LIN {X 0,Y 529.765,Z 572.438,A -85,B 0,C 180,E1 25488.601,E2 25488.601} C_VEL
LIN {X 0,Y 529.183,Z 585.576,A -85,B 0,C 180,E1 25486.804,E2 25486.804} C_VEL
LIN {X 0,Y 528.717,Z 597.375,A -85,B 0,C 180,E1 25484.904,E2 25484.904} C_VEL
LIN {X 0,Y 528.358,Z 608.331,A -85,B 0,C 180,E1 25482.792,E2 25482.792} C_VEL
LIN {X 0,Y 528.139,Z 617.247,A -85,B 0,C 180,E1 25480.693,E2 25480.693} C_VEL
LIN {X 0,Y 528.011,Z 624.374,A -85,B 0,C 180,E1 25478.604,E2 25478.604} C_VEL
LIN {X 0,Y 527.933,Z 630.003,A -85,B 0,C 180,E1 25476.416,E2 25476.416} C_VEL
LIN {X 0,Y 527.91,Z 633.928,A -85,B 0,C 180,E1 25474.237,E2 25474.237} C_VEL
LIN {X 0,Y 527.911,Z 636.306,A -85,B 0,C 180,E1 25471.954,E2 25471.954} C_VEL
LIN {X 0,Y 527.906,Z 636.962,A -85,B 0,C 180,E1 25469.784,E2 25469.784} C_VEL
LIN {X 0,Y 527.901,Z 636.034,A -85,B 0,C 180,E1 25467.613,E2 25467.613} C_VEL
LIN {X 0,Y 527.913,Z 633.45,A -85,B 0,C 180,E1 25465.438,E2 25465.438} C_VEL
LIN {X 0,Y 527.952,Z 629.246,A -85,B 0,C 180,E1 25463.258,E2 25463.258} C_VEL
LIN {X 0,Y 528.029,Z 623.329,A -85,B 0,C 180,E1 25461.068,E2 25461.068} C_VEL
LIN {X 0,Y 528.171,Z 616.015,A -85,B 0,C 180,E1 25458.978,E2 25458.978} C_VEL
LIN {X 0,Y 528.406,Z 606.785,A -85,B 0,C 180,E1 25456.876,E2 25456.876} C_VEL
LIN {X 0,Y 528.766,Z 596.111,A -85,B 0,C 180,E1 25454.874,E2 25454.874} C_VEL
LIN {X 0,Y 529.254,Z 583.72,A -85,B 0,C 180,E1 25452.926,E2 25452.926} C_VEL
LIN {X 0,Y 529.883,Z 569.672,A -85,B 0,C 180,E1 25451.062,E2 25451.062} C_VEL
LIN {X 0,Y 530.615,Z 554.618,A -85,B 0,C 180,E1 25449.368,E2 25449.368} C_VEL
LIN {X 0,Y 531.432,Z 538.622,A -85,B 0,C 180,E1 25447.839,E2 25447.839} C_VEL
LIN {X 0,Y 532.324,Z 520.994,A -85,B 0,C 180,E1 25446.418,E2 25446.418} C_VEL
LIN {X 0,Y 533.203,Z 502.232,A -85,B 0,C 180,E1 25445.164,E2 25445.164} C_VEL
LIN {X 0,Y 534.026,Z 483.351,A -85,B 0,C 180,E1 25444.136,E2 25444.136} C_VEL
LIN {X 0,Y 534.767,Z 464.127,A -85,B 0,C 180,E1 25443.301,E2 25443.301} C_VEL
LIN {X 0,Y 535.396,Z 443.369,A -85,B 0,C 180,E1 25442.614,E2 25442.614} C_VEL
LIN {X 0,Y 535.876,Z 422.691,A -85,B 0,C 180,E1 25442.142,E2 25442.142} C_VEL
LIN {X 0,Y 537.477,Z 229.841,A -85,B 0,C 180,E1 25439.341,E2 25439.341} C_VEL
LIN {X 0,Y 537.719,Z 174.211,A -85,B 0,C 180,E1 25438.529,E2 25438.529} C_VEL
LIN {X 0,Y 535.937,Z 162.685,A -85,B 0,C 180,E1 25438.227,E2 25438.227} C_VEL
LIN {X 0,Y 536.978,Z 125.392,A -85,B 0,C 180,E1 25435.72,E2 25435.72} C_VEL
LIN {X 0,Y 528.489,Z 103.658,A -85,B 0,C 180,E1 25433.555,E2 25433.555} C_VEL
LIN {X 0,Y 528.528,Z 103.65,A -85,B 0,C 180,E1 25430.18,E2 25430.18} C_VEL
LIN {X 0,Y 528.47,Z 103.654,A -85,B 0,C 180,E1 25426.912,E2 25426.912} C_VEL
LIN {X 0,Y 528.472,Z 103.65,A -85,B 0,C 180,E1 25423.406,E2 25423.406} C_VEL
LIN {X 0,Y 528.528,Z 103.639,A -85,B 0,C 180,E1 25420.159,E2 25420.159} C_VEL
LIN {X 0,Y 528.473,Z 103.643,A -85,B 0,C 180,E1 25416.842,E2 25416.842} C_VEL
LIN {X 0,Y 528.467,Z 103.648,A -85,B 0,C 180,E1 25413.406,E2 25413.406} C_VEL
LIN {X 0,Y 528.522,Z 103.651,A -85,B 0,C 180,E1 25410.088,E2 25410.088} C_VEL
LIN {X 0,Y 528.482,Z 103.651,A -85,B 0,C 180,E1 25406.75,E2 25406.75} C_VEL
LIN {X 0,Y 528.463,Z 103.649,A -85,B 0,C 180,E1 25403.411,E2 25403.411} C_VEL
LIN {X 0,Y 528.514,Z 103.648,A -85,B 0,C 180,E1 25400.14,E2 25400.14} C_VEL
LIN {X 0,Y 528.482,Z 103.65,A -85,B 0,C 180,E1 25396.803,E2 25396.803} C_VEL
LIN {X 0,Y 528.459,Z 103.644,A -85,B 0,C 180,E1 25393.457,E2 25393.457} C_VEL
LIN {X 0,Y 528.504,Z 103.654,A -85,B 0,C 180,E1 25390.133,E2 25390.133} C_VEL
LIN {X 0,Y 528.479,Z 103.643,A -85,B 0,C 180,E1 25386.845,E2 25386.845} C_VEL
LIN {X 0,Y 528.457,Z 103.653,A -85,B 0,C 180,E1 25383.471,E2 25383.471} C_VEL
LIN {X 0,Y 528.491,Z 103.65,A -85,B 0,C 180,E1 25380.108,E2 25380.108} C_VEL
LIN {X 0,Y 528.483,Z 103.653,A -85,B 0,C 180,E1 25376.855,E2 25376.855} C_VEL
LIN {X 0,Y 528.453,Z 103.65,A -85,B 0,C 180,E1 25373.59,E2 25373.59} C_VEL
LIN {X 0,Y 528.503,Z 103.65,A -85,B 0,C 180,E1 25370.306,E2 25370.306} C_VEL
LIN {X 0,Y 528.474,Z 103.648,A -85,B 0,C 180,E1 25366.988,E2 25366.988} C_VEL
LIN {X 0,Y 528.451,Z 103.65,A -85,B 0,C 180,E1 25363.625,E2 25363.625} C_VEL
LIN {X 0,Y 528.496,Z 103.655,A -85,B 0,C 180,E1 25360.32,E2 25360.32} C_VEL
LIN {X 0,Y 528.472,Z 103.649,A -85,B 0,C 180,E1 25357.061,E2 25357.061} C_VEL
LIN {X 0,Y 528.451,Z 103.654,A -85,B 0,C 180,E1 25353.721,E2 25353.721} C_VEL
LIN {X 0,Y 528.495,Z 103.653,A -85,B 0,C 180,E1 25350.41,E2 25350.41} C_VEL
LIN {X 0,Y 528.468,Z 103.651,A -85,B 0,C 180,E1 25347.143,E2 25347.143} C_VEL
LIN {X 0,Y 528.447,Z 103.654,A -85,B 0,C 180,E1 25343.82,E2 25343.82} C_VEL
LIN {X 0,Y 528.446,Z 103.654,A -85,B 0,C 180,E1 25341.679,E2 25341.679} C_VEL
LIN {X 0,Y 527.465,Z 103.785,A -85,B 0,C 180,E1 25340.844,E2 25340.844} C_VEL
LIN {X 0,Y 520.951,Z 104.593,A -85,B 0,C 180,E1 25338.436,E2 25338.436} C_VEL
LIN {X 0,Y 520.509,Z 104.645,A -85,B 0,C 180,E1 25337.885,E2 25337.885} C_VEL
LIN {X 0,Y 520.55,Z 104.646,A -85,B 0,C 180,E1 25334.513,E2 25334.513} C_VEL
LIN {X 0,Y 520.537,Z 104.646,A -85,B 0,C 180,E1 25331.152,E2 25331.152} C_VEL
LIN {X 0,Y 520.507,Z 104.643,A -85,B 0,C 180,E1 25327.789,E2 25327.789} C_VEL
LIN {X 0,Y 520.545,Z 104.646,A -85,B 0,C 180,E1 25324.51,E2 25324.51} C_VEL
LIN {X 0,Y 520.575,Z 104.775,A -85,B 0,C 180,E1 25323.04,E2 25323.04} C_VEL
LIN {X 0,Y 527.861,Z 125.987,A -85,B 0,C 180,E1 25320.537,E2 25320.537} C_VEL
LIN {X 0,Y 526.199,Z 167.004,A -85,B 0,C 180,E1 25316.978,E2 25316.978} C_VEL
LIN {X 0,Y 526.012,Z 175.066,A -85,B 0,C 180,E1 25316.321,E2 25316.321} C_VEL
LIN {X 0,Y 528.496,Z 189.23,A -85,B 0,C 180,E1 25315.966,E2 25315.966} C_VEL
LIN {X 0,Y 527.248,Z 386.361,A -85,B 0,C 180,E1 25313.208,E2 25313.208} C_VEL
LIN {X 0,Y 526.831,Z 405.219,A -85,B 0,C 180,E1 25312.735,E2 25312.735} C_VEL
LIN {X 0,Y 526.216,Z 423.519,A -85,B 0,C 180,E1 25312.06,E2 25312.06} C_VEL
LIN {X 0,Y 525.435,Z 441.08,A -85,B 0,C 180,E1 25311.195,E2 25311.195} C_VEL
LIN {X 0,Y 524.608,Z 457.322,A -85,B 0,C 180,E1 25310.179,E2 25310.179} C_VEL
LIN {X 0,Y 523.697,Z 473.407,A -85,B 0,C 180,E1 25308.939,E2 25308.939} C_VEL
LIN {X 0,Y 522.844,Z 487.847,A -85,B 0,C 180,E1 25307.586,E2 25307.586} C_VEL
LIN {X 0,Y 522.076,Z 500.906,A -85,B 0,C 180,E1 25306.122,E2 25306.122} C_VEL
LIN {X 0,Y 521.361,Z 513.526,A -85,B 0,C 180,E1 25304.422,E2 25304.422} C_VEL
LIN {X 0,Y 520.824,Z 524.475,A -85,B 0,C 180,E1 25302.641,E2 25302.641} C_VEL
LIN {X 0,Y 520.419,Z 534.066,A -85,B 0,C 180,E1 25300.74,E2 25300.74} C_VEL
LIN {X 0,Y 520.156,Z 542.149,A -85,B 0,C 180,E1 25298.734,E2 25298.734} C_VEL
LIN {X 0,Y 520.012,Z 548.653,A -85,B 0,C 180,E1 25296.624,E2 25296.624} C_VEL
LIN {X 0,Y 519.946,Z 553.265,A -85,B 0,C 180,E1 25294.521,E2 25294.521} C_VEL
LIN {X 0,Y 519.92,Z 556.105,A -85,B 0,C 180,E1 25292.424,E2 25292.424} C_VEL
LIN {X 0,Y 519.916,Z 557.244,A -85,B 0,C 180,E1 25290.33,E2 25290.33} C_VEL
LIN {X 0,Y 519.921,Z 556.706,A -85,B 0,C 180,E1 25288.236,E2 25288.236} C_VEL
LIN {X 0,Y 519.933,Z 554.482,A -85,B 0,C 180,E1 25286.14,E2 25286.14} C_VEL
LIN {X 0,Y 519.979,Z 550.762,A -85,B 0,C 180,E1 25284.15,E2 25284.15} C_VEL
LIN {X 0,Y 520.084,Z 545.397,A -85,B 0,C 180,E1 25282.154,E2 25282.154} C_VEL
LIN {X 0,Y 520.269,Z 538.258,A -85,B 0,C 180,E1 25280.151,E2 25280.151} C_VEL
LIN {X 0,Y 520.588,Z 529.681,A -85,B 0,C 180,E1 25278.253,E2 25278.253} C_VEL
LIN {X 0,Y 521.04,Z 519.746,A -85,B 0,C 180,E1 25276.46,E2 25276.46} C_VEL
LIN {X 0,Y 521.631,Z 508.493,A -85,B 0,C 180,E1 25274.775,E2 25274.775} C_VEL
LIN {X 0,Y 522.358,Z 495.896,A -85,B 0,C 180,E1 25273.199,E2 25273.199} C_VEL
LIN {X 0,Y 523.186,Z 481.855,A -85,B 0,C 180,E1 25271.734,E2 25271.734} C_VEL
LIN {X 0,Y 524.061,Z 466.923,A -85,B 0,C 180,E1 25270.443,E2 25270.443} C_VEL
LIN {X 0,Y 524.935,Z 450.956,A -85,B 0,C 180,E1 25269.308,E2 25269.308} C_VEL
LIN {X 0,Y 525.758,Z 434.164,A -85,B 0,C 180,E1 25268.349,E2 25268.349} C_VEL
LIN {X 0,Y 526.439,Z 417.282,A -85,B 0,C 180,E1 25267.598,E2 25267.598} C_VEL
LIN {X 0,Y 526.976,Z 398.776,A -85,B 0,C 180,E1 25266.992,E2 25266.992} C_VEL
LIN {X 0,Y 527.313,Z 379.889,A -85,B 0,C 180,E1 25266.591,E2 25266.591} C_VEL
LIN {X 0,Y 528.392,Z 187.436,A -85,B 0,C 180,E1 25263.911,E2 25263.911} C_VEL
LIN {X 0,Y 525.938,Z 174.407,A -85,B 0,C 180,E1 25263.563,E2 25263.563} C_VEL
LIN {X 0,Y 527.535,Z 134.94,A -85,B 0,C 180,E1 25260.163,E2 25260.163} C_VEL
LIN {X 0,Y 527.776,Z 125.562,A -85,B 0,C 180,E1 25259.327,E2 25259.327} C_VEL
LIN {X 0,Y 520.548,Z 104.642,A -85,B 0,C 180,E1 25256.845,E2 25256.845} C_VEL
LIN {X 0,Y 520.584,Z 104.646,A -85,B 0,C 180,E1 25253.458,E2 25253.458} C_VEL
LIN {X 0,Y 520.556,Z 104.626,A -85,B 0,C 180,E1 25250.03,E2 25250.03} C_VEL
LIN {X 0,Y 520.557,Z 104.637,A -85,B 0,C 180,E1 25246.708,E2 25246.708} C_VEL
LIN {X 0,Y 520.584,Z 104.633,A -85,B 0,C 180,E1 25243.287,E2 25243.287} C_VEL
LIN {X 0,Y 520.577,Z 104.639,A -85,B 0,C 180,E1 25239.801,E2 25239.801} C_VEL
LIN {X 0,Y 520.584,Z 104.642,A -85,B 0,C 180,E1 25236.405,E2 25236.405} C_VEL
LIN {X 0,Y 520.585,Z 104.64,A -85,B 0,C 180,E1 25232.925,E2 25232.925} C_VEL
LIN {X 0,Y 520.582,Z 104.769,A -85,B 0,C 180,E1 25232.24,E2 25232.24} C_VEL
LIN {X 0,Y 526.534,Z 123.353,A -85,B 0,C 180,E1 25230.34,E2 25230.34} C_VEL
LIN {X 0,Y 525.7,Z 163.174,A -85,B 0,C 180,E1 25227.111,E2 25227.111} C_VEL
LIN {X 0,Y 525.503,Z 178.656,A -85,B 0,C 180,E1 25225.886,E2 25225.886} C_VEL
LIN {X 0,Y 526.984,Z 189.32,A -85,B 0,C 180,E1 25225.642,E2 25225.642} C_VEL
LIN {X 0,Y 525.173,Z 387.373,A -85,B 0,C 180,E1 25222.681,E2 25222.681} C_VEL
LIN {X 0,Y 524.856,Z 406.213,A -85,B 0,C 180,E1 25222.201,E2 25222.201} C_VEL
LIN {X 0,Y 524.408,Z 424.605,A -85,B 0,C 180,E1 25221.527,E2 25221.527} C_VEL
LIN {X 0,Y 523.865,Z 442.073,A -85,B 0,C 180,E1 25220.677,E2 25220.677} C_VEL
LIN {X 0,Y 523.269,Z 458.726,A -85,B 0,C 180,E1 25219.652,E2 25219.652} C_VEL
LIN {X 0,Y 522.646,Z 474.476,A -85,B 0,C 180,E1 25218.458,E2 25218.458} C_VEL
LIN {X 0,Y 522.033,Z 489.163,A -85,B 0,C 180,E1 25217.109,E2 25217.109} C_VEL
LIN {X 0,Y 521.497,Z 502.095,A -85,B 0,C 180,E1 25215.685,E2 25215.685} C_VEL
LIN {X 0,Y 521.013,Z 514.069,A -85,B 0,C 180,E1 25214.107,E2 25214.107} C_VEL
LIN {X 0,Y 520.623,Z 524.698,A -85,B 0,C 180,E1 25212.421,E2 25212.421} C_VEL
LIN {X 0,Y 520.327,Z 533.934,A -85,B 0,C 180,E1 25210.631,E2 25210.631} C_VEL
LIN {X 0,Y 520.131,Z 541.822,A -85,B 0,C 180,E1 25208.735,E2 25208.735} C_VEL
LIN {X 0,Y 520.008,Z 548.485,A -85,B 0,C 180,E1 25206.625,E2 25206.625} C_VEL
LIN {X 0,Y 519.944,Z 553.013,A -85,B 0,C 180,E1 25204.633,E2 25204.633} C_VEL
LIN {X 0,Y 519.925,Z 556.084,A -85,B 0,C 180,E1 25202.425,E2 25202.425} C_VEL
LIN {X 0,Y 519.924,Z 557.231,A -85,B 0,C 180,E1 25200.441,E2 25200.441} C_VEL
LIN {X 0,Y 519.917,Z 556.723,A -85,B 0,C 180,E1 25198.237,E2 25198.237} C_VEL
LIN {X 0,Y 519.936,Z 554.631,A -85,B 0,C 180,E1 25196.251,E2 25196.251} C_VEL
LIN {X 0,Y 519.975,Z 550.755,A -85,B 0,C 180,E1 25194.151,E2 25194.151} C_VEL
LIN {X 0,Y 520.07,Z 545.259,A -85,B 0,C 180,E1 25192.155,E2 25192.155} C_VEL
LIN {X 0,Y 520.242,Z 537.967,A -85,B 0,C 180,E1 25190.151,E2 25190.151} C_VEL
LIN {X 0,Y 520.509,Z 529.084,A -85,B 0,C 180,E1 25188.252,E2 25188.252} C_VEL
LIN {X 0,Y 520.881,Z 518.649,A -85,B 0,C 180,E1 25186.457,E2 25186.457} C_VEL
LIN {X 0,Y 521.345,Z 506.639,A -85,B 0,C 180,E1 25184.767,E2 25184.767} C_VEL
LIN {X 0,Y 521.876,Z 493.512,A -85,B 0,C 180,E1 25183.242,E2 25183.242} C_VEL
LIN {X 0,Y 522.437,Z 479.395,A -85,B 0,C 180,E1 25181.881,E2 25181.881} C_VEL
LIN {X 0,Y 522.995,Z 464.402,A -85,B 0,C 180,E1 25180.687,E2 25180.687} C_VEL
LIN {X 0,Y 523.549,Z 447.666,A -85,B 0,C 180,E1 25179.603,E2 25179.603} C_VEL
LIN {X 0,Y 524.042,Z 429.772,A -85,B 0,C 180,E1 25178.687,E2 25178.687} C_VEL
LIN {X 0,Y 524.442,Z 411.447,A -85,B 0,C 180,E1 25177.977,E2 25177.977} C_VEL
LIN {X 0,Y 524.718,Z 392.774,A -85,B 0,C 180,E1 25177.465,E2 25177.465} C_VEL
LIN {X 0,Y 524.898,Z 369.628,A -85,B 0,C 180,E1 25177.08,E2 25177.08} C_VEL
LIN {X 0,Y 526.071,Z 235.724,A -85,B 0,C 180,E1 25175.092,E2 25175.092} C_VEL
LIN {X 0,Y 526.503,Z 186.515,A -85,B 0,C 180,E1 25174.299,E2 25174.299} C_VEL
LIN {X 0,Y 525.718,Z 181.291,A -85,B 0,C 180,E1 25174.148,E2 25174.148} C_VEL
LIN {X 0,Y 525.983,Z 146.706,A -85,B 0,C 180,E1 25171.502,E2 25171.502} C_VEL
LIN {X 0,Y 525.808,Z 121.117,A -85,B 0,C 180,E1 25169.594,E2 25169.594} C_VEL
LIN {X 0,Y 521.519,Z 107.586,A -85,B 0,C 180,E1 25168.347,E2 25168.347} C_VEL
LIN {X 0,Y 520.559,Z 104.644,A -85,B 0,C 180,E1 25168.051,E2 25168.051} C_VEL
LIN {X 0,Y 520.543,Z 104.644,A -85,B 0,C 180,E1 25164.679,E2 25164.679} C_VEL
LIN {X 0,Y 520.581,Z 104.644,A -85,B 0,C 180,E1 25161.376,E2 25161.376} C_VEL
LIN {X 0,Y 520.555,Z 104.643,A -85,B 0,C 180,E1 25158.017,E2 25158.017} C_VEL
LIN {X 0,Y 520.518,Z 104.646,A -85,B 0,C 180,E1 25154.673,E2 25154.673} C_VEL
LIN {X 0,Y 520.532,Z 104.647,A -85,B 0,C 180,E1 25151.319,E2 25151.319} C_VEL
LIN {X 0,Y 520.56,Z 104.645,A -85,B 0,C 180,E1 25148.048,E2 25148.048} C_VEL
LIN {X 0,Y 520.525,Z 104.695,A -85,B 0,C 180,E1 25146.958,E2 25146.958} C_VEL
LIN {X 0,Y 529.855,Z 128.471,A -85,B 0,C 180,E1 25144.544,E2 25144.544} C_VEL
LIN {X 0,Y 528.828,Z 163.796,A -85,B 0,C 180,E1 25142.157,E2 25142.157} C_VEL
LIN {X 0,Y 530.859,Z 178.032,A -85,B 0,C 180,E1 25141.813,E2 25141.813} C_VEL
LIN {X 0,Y 528.972,Z 409.172,A -85,B 0,C 180,E1 25138.479,E2 25138.479} C_VEL
LIN {X 0,Y 528.577,Z 432.03,A -85,B 0,C 180,E1 25138.074,E2 25138.074} C_VEL
LIN {X 0,Y 527.978,Z 453.124,A -85,B 0,C 180,E1 25137.487,E2 25137.487} C_VEL
LIN {X 0,Y 527.251,Z 472.243,A -85,B 0,C 180,E1 25136.763,E2 25136.763} C_VEL
LIN {X 0,Y 526.416,Z 491.221,A -85,B 0,C 180,E1 25135.843,E2 25135.843} C_VEL
LIN {X 0,Y 525.438,Z 510.314,A -85,B 0,C 180,E1 25134.689,E2 25134.689} C_VEL
LIN {X 0,Y 524.442,Z 528.371,A -85,B 0,C 180,E1 25133.364,E2 25133.364} C_VEL
LIN {X 0,Y 523.477,Z 545.423,A -85,B 0,C 180,E1 25131.868,E2 25131.868} C_VEL
LIN {X 0,Y 522.601,Z 561.226,A -85,B 0,C 180,E1 25130.227,E2 25130.227} C_VEL
LIN {X 0,Y 521.829,Z 575.9,A -85,B 0,C 180,E1 25128.431,E2 25128.431} C_VEL
LIN {X 0,Y 521.22,Z 588.57,A -85,B 0,C 180,E1 25126.609,E2 25126.609} C_VEL
LIN {X 0,Y 520.716,Z 600.533,A -85,B 0,C 180,E1 25124.569,E2 25124.569} C_VEL
LIN {X 0,Y 520.354,Z 610.902,A -85,B 0,C 180,E1 25122.428,E2 25122.428} C_VEL
LIN {X 0,Y 520.124,Z 619.273,A -85,B 0,C 180,E1 25120.299,E2 25120.299} C_VEL
LIN {X 0,Y 519.999,Z 625.896,A -85,B 0,C 180,E1 25118.181,E2 25118.181} C_VEL
LIN {X 0,Y 519.936,Z 631.14,A -85,B 0,C 180,E1 25115.961,E2 25115.961} C_VEL
LIN {X 0,Y 519.915,Z 634.709,A -85,B 0,C 180,E1 25113.75,E2 25113.75} C_VEL
LIN {X 0,Y 519.902,Z 636.575,A -85,B 0,C 180,E1 25111.544,E2 25111.544} C_VEL
LIN {X 0,Y 519.903,Z 636.873,A -85,B 0,C 180,E1 25109.34,E2 25109.34} C_VEL
LIN {X 0,Y 519.914,Z 635.507,A -85,B 0,C 180,E1 25107.024,E2 25107.024} C_VEL
LIN {X 0,Y 519.924,Z 632.583,A -85,B 0,C 180,E1 25104.815,E2 25104.815} C_VEL
LIN {X 0,Y 519.971,Z 627.975,A -85,B 0,C 180,E1 25102.598,E2 25102.598} C_VEL
LIN {X 0,Y 520.069,Z 621.915,A -85,B 0,C 180,E1 25100.484,E2 25100.484} C_VEL
LIN {X 0,Y 520.261,Z 613.722,A -85,B 0,C 180,E1 25098.247,E2 25098.247} C_VEL
LIN {X 0,Y 520.574,Z 603.993,A -85,B 0,C 180,E1 25096.109,E2 25096.109} C_VEL
LIN {X 0,Y 521.032,Z 592.791,A -85,B 0,C 180,E1 25094.074,E2 25094.074} C_VEL
LIN {X 0,Y 521.625,Z 580.137,A -85,B 0,C 180,E1 25092.141,E2 25092.141} C_VEL
LIN {X 0,Y 522.388,Z 565.491,A -85,B 0,C 180,E1 25090.257,E2 25090.257} C_VEL
LIN {X 0,Y 523.273,Z 549.462,A -85,B 0,C 180,E1 25088.52,E2 25088.52} C_VEL
LIN {X 0,Y 524.216,Z 532.618,A -85,B 0,C 180,E1 25086.984,E2 25086.984} C_VEL
LIN {X 0,Y 525.133,Z 515.658,A -85,B 0,C 180,E1 25085.681,E2 25085.681} C_VEL
LIN {X 0,Y 526.088,Z 497.286,A -85,B 0,C 180,E1 25084.503,E2 25084.503} C_VEL
LIN {X 0,Y 526.984,Z 478.563,A -85,B 0,C 180,E1 25083.522,E2 25083.522} C_VEL
LIN {X 0,Y 527.786,Z 458.777,A -85,B 0,C 180,E1 25082.701,E2 25082.701} C_VEL
LIN {X 0,Y 528.467,Z 437.999,A -85,B 0,C 180,E1 25082.067,E2 25082.067} C_VEL
LIN {X 0,Y 528.872,Z 417.592,A -85,B 0,C 180,E1 25081.649,E2 25081.649} C_VEL
LIN {X 0,Y 530.786,Z 185.26,A -85,B 0,C 180,E1 25078.293,E2 25078.293} C_VEL
LIN {X 0,Y 530.645,Z 175.238,A -85,B 0,C 180,E1 25078.131,E2 25078.131} C_VEL
LIN {X 0,Y 528.759,Z 162.912,A -85,B 0,C 180,E1 25077.808,E2 25077.808} C_VEL
LIN {X 0,Y 529.858,Z 128.465,A -85,B 0,C 180,E1 25075.456,E2 25075.456} C_VEL
LIN {X 0,Y 521.321,Z 107.242,A -85,B 0,C 180,E1 25073.292,E2 25073.292} C_VEL
LIN {X 0,Y 520.532,Z 104.646,A -85,B 0,C 180,E1 25073.013,E2 25073.013} C_VEL
LIN {X 0,Y 520.555,Z 104.643,A -85,B 0,C 180,E1 25069.663,E2 25069.663} C_VEL
LIN {X 0,Y 520.583,Z 104.638,A -85,B 0,C 180,E1 25066.233,E2 25066.233} C_VEL
LIN {X 0,Y 520.531,Z 104.638,A -85,B 0,C 180,E1 25062.96,E2 25062.96} C_VEL
LIN {X 0,Y 520.531,Z 104.623,A -85,B 0,C 180,E1 25059.452,E2 25059.452} C_VEL
LIN {X 0,Y 520.581,Z 104.633,A -85,B 0,C 180,E1 25056.131,E2 25056.131} C_VEL
LIN {X 0,Y 520.537,Z 104.635,A -85,B 0,C 180,E1 25052.797,E2 25052.797} C_VEL
LIN {X 0,Y 520.529,Z 104.638,A -85,B 0,C 180,E1 25049.455,E2 25049.455} C_VEL
LIN {X 0,Y 520.583,Z 104.642,A -85,B 0,C 180,E1 25046.215,E2 25046.215} C_VEL
LIN {X 0,Y 520.538,Z 104.637,A -85,B 0,C 180,E1 25042.83,E2 25042.83} C_VEL
LIN {X 0,Y 520.522,Z 104.635,A -85,B 0,C 180,E1 25039.409,E2 25039.409} C_VEL
LIN {X 0,Y 520.563,Z 104.643,A -85,B 0,C 180,E1 25036.056,E2 25036.056} C_VEL
LIN {X 0,Y 520.536,Z 104.631,A -85,B 0,C 180,E1 25032.874,E2 25032.874} C_VEL
LIN {X 0,Y 520.521,Z 104.642,A -85,B 0,C 180,E1 25029.508,E2 25029.508} C_VEL
LIN {X 0,Y 520.565,Z 104.636,A -85,B 0,C 180,E1 25026.174,E2 25026.174} C_VEL
LIN {X 0,Y 520.545,Z 104.642,A -85,B 0,C 180,E1 25022.816,E2 25022.816} C_VEL
LIN {X 0,Y 520.517,Z 104.64,A -85,B 0,C 180,E1 25019.449,E2 25019.449} C_VEL
LIN {X 0,Y 520.551,Z 104.637,A -85,B 0,C 180,E1 25016.145,E2 25016.145} C_VEL
LIN {X 0,Y 520.548,Z 104.637,A -85,B 0,C 180,E1 25012.828,E2 25012.828} C_VEL
LIN {X 0,Y 520.514,Z 104.638,A -85,B 0,C 180,E1 25009.485,E2 25009.485} C_VEL
LIN {X 0,Y 520.539,Z 104.644,A -85,B 0,C 180,E1 25006.107,E2 25006.107} C_VEL
LIN {X 0,Y 520.543,Z 104.638,A -85,B 0,C 180,E1 25002.909,E2 25002.909} C_VEL
LIN {X 0,Y 520.512,Z 104.643,A -85,B 0,C 180,E1 24999.537,E2 24999.537} C_VEL
LIN {X 0,Y 520.54,Z 104.639,A -85,B 0,C 180,E1 24996.211,E2 24996.211} C_VEL
LIN {X 0,Y 520.548,Z 104.642,A -85,B 0,C 180,E1 24992.92,E2 24992.92} C_VEL
LIN {X 0,Y 520.508,Z 104.643,A -85,B 0,C 180,E1 24989.596,E2 24989.596} C_VEL
LIN {X 0,Y 520.537,Z 104.642,A -85,B 0,C 180,E1 24986.274,E2 24986.274} C_VEL
LIN {X 0,Y 520.554,Z 104.639,A -85,B 0,C 180,E1 24982.906,E2 24982.906} C_VEL
LIN {X 0,Y 520.507,Z 104.643,A -85,B 0,C 180,E1 24979.657,E2 24979.657} C_VEL
LIN {X 0,Y 520.509,Z 104.645,A -85,B 0,C 180,E1 24977.885,E2 24977.885} C_VEL
LIN {X 0,Y 519.522,Z 104.774,A -85,B 0,C 180,E1 24977.038,E2 24977.038} C_VEL
LIN {X 0,Y 513.028,Z 105.583,A -85,B 0,C 180,E1 24974.593,E2 24974.593} C_VEL
LIN {X 0,Y 512.574,Z 105.635,A -85,B 0,C 180,E1 24974.034,E2 24974.034} C_VEL
LIN {X 0,Y 512.626,Z 105.629,A -85,B 0,C 180,E1 24970.647,E2 24970.647} C_VEL
LIN {X 0,Y 512.585,Z 105.632,A -85,B 0,C 180,E1 24967.346,E2 24967.346} C_VEL
LIN {X 0,Y 512.571,Z 105.639,A -85,B 0,C 180,E1 24963.909,E2 24963.909} C_VEL
LIN {X 0,Y 512.583,Z 105.698,A -85,B 0,C 180,E1 24963.579,E2 24963.579} C_VEL
LIN {X 0,Y 520.525,Z 128.355,A -85,B 0,C 180,E1 24960.837,E2 24960.837} C_VEL
LIN {X 0,Y 519.59,Z 151.742,A -85,B 0,C 180,E1 24958.755,E2 24958.755} C_VEL
LIN {X 0,Y 518.738,Z 174.94,A -85,B 0,C 180,E1 24956.774,E2 24956.774} C_VEL
LIN {X 0,Y 521.49,Z 190.46,A -85,B 0,C 180,E1 24956.375,E2 24956.375} C_VEL
LIN {X 0,Y 520.219,Z 386.818,A -85,B 0,C 180,E1 24953.623,E2 24953.623} C_VEL
LIN {X 0,Y 519.777,Z 405.786,A -85,B 0,C 180,E1 24953.145,E2 24953.145} C_VEL
LIN {X 0,Y 519.128,Z 423.825,A -85,B 0,C 180,E1 24952.476,E2 24952.476} C_VEL
LIN {X 0,Y 518.303,Z 441.142,A -85,B 0,C 180,E1 24951.62,E2 24951.62} C_VEL
LIN {X 0,Y 517.391,Z 457.503,A -85,B 0,C 180,E1 24950.591,E2 24950.591} C_VEL
LIN {X 0,Y 516.367,Z 473.626,A -85,B 0,C 180,E1 24949.335,E2 24949.335} C_VEL
LIN {X 0,Y 515.396,Z 488.088,A -85,B 0,C 180,E1 24947.965,E2 24947.965} C_VEL
LIN {X 0,Y 514.456,Z 502.06,A -85,B 0,C 180,E1 24946.367,E2 24946.367} C_VEL
LIN {X 0,Y 513.66,Z 514.486,A -85,B 0,C 180,E1 24944.657,E2 24944.657} C_VEL
LIN {X 0,Y 513.039,Z 525.428,A -85,B 0,C 180,E1 24942.836,E2 24942.836} C_VEL
LIN {X 0,Y 512.563,Z 534.918,A -85,B 0,C 180,E1 24940.906,E2 24940.906} C_VEL
LIN {X 0,Y 512.247,Z 542.921,A -85,B 0,C 180,E1 24938.87,E2 24938.87} C_VEL
LIN {X 0,Y 512.072,Z 549.367,A -85,B 0,C 180,E1 24936.727,E2 24936.727} C_VEL
LIN {X 0,Y 511.986,Z 553.943,A -85,B 0,C 180,E1 24934.592,E2 24934.592} C_VEL
LIN {X 0,Y 511.95,Z 556.76,A -85,B 0,C 180,E1 24932.462,E2 24932.462} C_VEL
LIN {X 0,Y 511.942,Z 557.889,A -85,B 0,C 180,E1 24930.335,E2 24930.335} C_VEL
LIN {X 0,Y 511.949,Z 557.356,A -85,B 0,C 180,E1 24928.209,E2 24928.209} C_VEL
LIN {X 0,Y 511.969,Z 555.151,A -85,B 0,C 180,E1 24926.08,E2 24926.08} C_VEL
LIN {X 0,Y 512.036,Z 551.217,A -85,B 0,C 180,E1 24923.946,E2 24923.946} C_VEL
LIN {X 0,Y 512.168,Z 545.8,A -85,B 0,C 180,E1 24921.919,E2 24921.919} C_VEL
LIN {X 0,Y 512.409,Z 538.621,A -85,B 0,C 180,E1 24919.885,E2 24919.885} C_VEL
LIN {X 0,Y 512.795,Z 530.021,A -85,B 0,C 180,E1 24917.957,E2 24917.957} C_VEL
LIN {X 0,Y 513.331,Z 520.061,A -85,B 0,C 180,E1 24916.138,E2 24916.138} C_VEL
LIN {X 0,Y 514.016,Z 508.775,A -85,B 0,C 180,E1 24914.428,E2 24914.428} C_VEL
LIN {X 0,Y 514.847,Z 496.132,A -85,B 0,C 180,E1 24912.83,E2 24912.83} C_VEL
LIN {X 0,Y 515.791,Z 482.067,A -85,B 0,C 180,E1 24911.345,E2 24911.345} C_VEL
LIN {X 0,Y 516.734,Z 467.738,A -85,B 0,C 180,E1 24910.089,E2 24910.089} C_VEL
LIN {X 0,Y 517.696,Z 451.932,A -85,B 0,C 180,E1 24908.946,E2 24908.946} C_VEL
LIN {X 0,Y 518.594,Z 435.251,A -85,B 0,C 180,E1 24907.977,E2 24907.977} C_VEL
LIN {X 0,Y 519.374,Z 417.417,A -85,B 0,C 180,E1 24907.175,E2 24907.175} C_VEL
LIN {X 0,Y 519.938,Z 399.145,A -85,B 0,C 180,E1 24906.576,E2 24906.576} C_VEL
LIN {X 0,Y 520.28,Z 380.548,A -85,B 0,C 180,E1 24906.18,E2 24906.18} C_VEL
LIN {X 0,Y 521.371,Z 188.643,A -85,B 0,C 180,E1 24903.5,E2 24903.5} C_VEL
LIN {X 0,Y 518.668,Z 174.395,A -85,B 0,C 180,E1 24903.118,E2 24903.118} C_VEL
LIN {X 0,Y 520.401,Z 135.373,A -85,B 0,C 180,E1 24899.711,E2 24899.711} C_VEL
LIN {X 0,Y 520.477,Z 128.198,A -85,B 0,C 180,E1 24899.054,E2 24899.054} C_VEL
LIN {X 0,Y 513.463,Z 108.384,A -85,B 0,C 180,E1 24896.656,E2 24896.656} C_VEL
LIN {X 0,Y 512.586,Z 105.633,A -85,B 0,C 180,E1 24896.292,E2 24896.292} C_VEL
LIN {X 0,Y 512.62,Z 105.634,A -85,B 0,C 180,E1 24892.916,E2 24892.916} C_VEL
LIN {X 0,Y 512.651,Z 105.619,A -85,B 0,C 180,E1 24889.497,E2 24889.497} C_VEL
LIN {X 0,Y 512.638,Z 105.627,A -85,B 0,C 180,E1 24886.024,E2 24886.024} C_VEL
LIN {X 0,Y 512.63,Z 105.626,A -85,B 0,C 180,E1 24882.5,E2 24882.5} C_VEL
LIN {X 0,Y 512.64,Z 105.626,A -85,B 0,C 180,E1 24879.049,E2 24879.049} C_VEL
LIN {X 0,Y 512.638,Z 105.628,A -85,B 0,C 180,E1 24875.537,E2 24875.537} C_VEL
LIN {X 0,Y 512.663,Z 105.754,A -85,B 0,C 180,E1 24872.667,E2 24872.667} C_VEL
LIN {X 0,Y 519.209,Z 126.108,A -85,B 0,C 180,E1 24870.557,E2 24870.557} C_VEL
LIN {X 0,Y 518.307,Z 165.689,A -85,B 0,C 180,E1 24867.331,E2 24867.331} C_VEL
LIN {X 0,Y 518.138,Z 179.197,A -85,B 0,C 180,E1 24866.262,E2 24866.262} C_VEL
LIN {X 0,Y 519.721,Z 190.473,A -85,B 0,C 180,E1 24865.998,E2 24865.998} C_VEL
LIN {X 0,Y 517.659,Z 388.199,A -85,B 0,C 180,E1 24862.974,E2 24862.974} C_VEL
LIN {X 0,Y 517.309,Z 407.426,A -85,B 0,C 180,E1 24862.471,E2 24862.471} C_VEL
LIN {X 0,Y 516.819,Z 425.823,A -85,B 0,C 180,E1 24861.777,E2 24861.777} C_VEL
LIN {X 0,Y 516.208,Z 443.742,A -85,B 0,C 180,E1 24860.879,E2 24860.879} C_VEL
LIN {X 0,Y 515.569,Z 460.187,A -85,B 0,C 180,E1 24859.84,E2 24859.84} C_VEL
LIN {X 0,Y 514.897,Z 475.85,A -85,B 0,C 180,E1 24858.624,E2 24858.624} C_VEL
LIN {X 0,Y 514.235,Z 490.472,A -85,B 0,C 180,E1 24857.249,E2 24857.249} C_VEL
LIN {X 0,Y 513.617,Z 504.128,A -85,B 0,C 180,E1 24855.7,E2 24855.7} C_VEL
LIN {X 0,Y 513.068,Z 516.851,A -85,B 0,C 180,E1 24853.952,E2 24853.952} C_VEL
LIN {X 0,Y 512.651,Z 527.557,A -85,B 0,C 180,E1 24852.16,E2 24852.16} C_VEL
LIN {X 0,Y 512.349,Z 536.411,A -85,B 0,C 180,E1 24850.343,E2 24850.343} C_VEL
LIN {X 0,Y 512.146,Z 543.896,A -85,B 0,C 180,E1 24848.42,E2 24848.42} C_VEL
LIN {X 0,Y 512.034,Z 549.931,A -85,B 0,C 180,E1 24846.391,E2 24846.391} C_VEL
LIN {X 0,Y 511.968,Z 554.211,A -85,B 0,C 180,E1 24844.368,E2 24844.368} C_VEL
LIN {X 0,Y 511.954,Z 556.955,A -85,B 0,C 180,E1 24842.239,E2 24842.239} C_VEL
LIN {X 0,Y 511.95,Z 557.964,A -85,B 0,C 180,E1 24840.112,E2 24840.112} C_VEL
LIN {X 0,Y 511.95,Z 557.263,A -85,B 0,C 180,E1 24837.986,E2 24837.986} C_VEL
LIN {X 0,Y 511.972,Z 554.85,A -85,B 0,C 180,E1 24835.856,E2 24835.856} C_VEL
LIN {X 0,Y 512.04,Z 550.614,A -85,B 0,C 180,E1 24833.722,E2 24833.722} C_VEL
LIN {X 0,Y 512.147,Z 544.812,A -85,B 0,C 180,E1 24831.694,E2 24831.694} C_VEL
LIN {X 0,Y 512.358,Z 537.568,A -85,B 0,C 180,E1 24829.771,E2 24829.771} C_VEL
LIN {X 0,Y 512.648,Z 528.964,A -85,B 0,C 180,E1 24827.955,E2 24827.955} C_VEL
LIN {X 0,Y 513.065,Z 518.293,A -85,B 0,C 180,E1 24826.131,E2 24826.131} C_VEL
LIN {X 0,Y 513.549,Z 506.887,A -85,B 0,C 180,E1 24824.526,E2 24824.526} C_VEL
LIN {X 0,Y 514.122,Z 493.645,A -85,B 0,C 180,E1 24822.981,E2 24822.981} C_VEL
LIN {X 0,Y 514.756,Z 478.683,A -85,B 0,C 180,E1 24821.542,E2 24821.542} C_VEL
LIN {X 0,Y 515.361,Z 463.306,A -85,B 0,C 180,E1 24820.33,E2 24820.33} C_VEL
LIN {X 0,Y 515.926,Z 447.071,A -85,B 0,C 180,E1 24819.287,E2 24819.287} C_VEL
LIN {X 0,Y 516.44,Z 429.349,A -85,B 0,C 180,E1 24818.384,E2 24818.384} C_VEL
LIN {X 0,Y 516.854,Z 410.997,A -85,B 0,C 180,E1 24817.677,E2 24817.677} C_VEL
LIN {X 0,Y 517.146,Z 391.898,A -85,B 0,C 180,E1 24817.162,E2 24817.162} C_VEL
LIN {X 0,Y 517.411,Z 356.715,A -85,B 0,C 180,E1 24816.611,E2 24816.611} C_VEL
LIN {X 0,Y 518.785,Z 230.993,A -85,B 0,C 180,E1 24814.668,E2 24814.668} C_VEL
LIN {X 0,Y 519.266,Z 187.724,A -85,B 0,C 180,E1 24813.943,E2 24813.943} C_VEL
LIN {X 0,Y 518.466,Z 182.523,A -85,B 0,C 180,E1 24813.793,E2 24813.793} C_VEL
LIN {X 0,Y 518.76,Z 146.987,A -85,B 0,C 180,E1 24811.068,E2 24811.068} C_VEL
LIN {X 0,Y 518.558,Z 123.625,A -85,B 0,C 180,E1 24809.312,E2 24809.312} C_VEL
LIN {X 0,Y 514.525,Z 111.129,A -85,B 0,C 180,E1 24808.126,E2 24808.126} C_VEL
LIN {X 0,Y 512.649,Z 105.632,A -85,B 0,C 180,E1 24807.564,E2 24807.564} C_VEL
LIN {X 0,Y 512.609,Z 105.632,A -85,B 0,C 180,E1 24804.186,E2 24804.186} C_VEL
LIN {X 0,Y 512.596,Z 105.634,A -85,B 0,C 180,E1 24800.75,E2 24800.75} C_VEL
LIN {X 0,Y 512.627,Z 105.634,A -85,B 0,C 180,E1 24797.405,E2 24797.405} C_VEL
LIN {X 0,Y 512.618,Z 105.633,A -85,B 0,C 180,E1 24793.968,E2 24793.968} C_VEL
LIN {X 0,Y 512.573,Z 105.636,A -85,B 0,C 180,E1 24790.641,E2 24790.641} C_VEL
LIN {X 0,Y 512.644,Z 105.877,A -85,B 0,C 180,E1 24787.483,E2 24787.483} C_VEL
LIN {X 0,Y 522.756,Z 131.839,A -85,B 0,C 180,E1 24784.794,E2 24784.794} C_VEL
LIN {X 0,Y 521.666,Z 163.819,A -85,B 0,C 180,E1 24782.598,E2 24782.598} C_VEL
LIN {X 0,Y 523.844,Z 179.287,A -85,B 0,C 180,E1 24782.218,E2 24782.218} C_VEL
LIN {X 0,Y 521.695,Z 404.616,A -85,B 0,C 180,E1 24778.9,E2 24778.9} C_VEL
LIN {X 0,Y 521.294,Z 430.959,A -85,B 0,C 180,E1 24778.454,E2 24778.454} C_VEL
LIN {X 0,Y 520.695,Z 452.593,A -85,B 0,C 180,E1 24777.87,E2 24777.87} C_VEL
LIN {X 0,Y 519.999,Z 471.567,A -85,B 0,C 180,E1 24777.171,E2 24777.171} C_VEL
LIN {X 0,Y 519.245,Z 488.95,A -85,B 0,C 180,E1 24776.35,E2 24776.35} C_VEL
LIN {X 0,Y 518.233,Z 506.846,A -85,B 0,C 180,E1 24775.291,E2 24775.291} C_VEL
LIN {X 0,Y 517.146,Z 525.429,A -85,B 0,C 180,E1 24773.956,E2 24773.956} C_VEL
LIN {X 0,Y 516.145,Z 541.773,A -85,B 0,C 180,E1 24772.555,E2 24772.555} C_VEL
LIN {X 0,Y 515.148,Z 557.885,A -85,B 0,C 180,E1 24770.925,E2 24770.925} C_VEL
LIN {X 0,Y 514.22,Z 573.353,A -85,B 0,C 180,E1 24769.067,E2 24769.067} C_VEL
LIN {X 0,Y 513.443,Z 587.58,A -85,B 0,C 180,E1 24767.03,E2 24767.03} C_VEL
LIN {X 0,Y 512.867,Z 599.278,A -85,B 0,C 180,E1 24765.029,E2 24765.029} C_VEL
LIN {X 0,Y 512.453,Z 609.358,A -85,B 0,C 180,E1 24762.967,E2 24762.967} C_VEL
LIN {X 0,Y 512.183,Z 618.058,A -85,B 0,C 180,E1 24760.802,E2 24760.802} C_VEL
LIN {X 0,Y 512.027,Z 624.986,A -85,B 0,C 180,E1 24758.649,E2 24758.649} C_VEL
LIN {X 0,Y 511.939,Z 630.507,A -85,B 0,C 180,E1 24756.392,E2 24756.392} C_VEL
LIN {X 0,Y 511.914,Z 634.245,A -85,B 0,C 180,E1 24754.145,E2 24754.145} C_VEL
LIN {X 0,Y 511.909,Z 636.373,A -85,B 0,C 180,E1 24751.904,E2 24751.904} C_VEL
LIN {X 0,Y 511.9,Z 636.918,A -85,B 0,C 180,E1 24749.553,E2 24749.553} C_VEL
LIN {X 0,Y 511.908,Z 635.843,A -85,B 0,C 180,E1 24747.314,E2 24747.314} C_VEL
LIN {X 0,Y 511.927,Z 633.129,A -85,B 0,C 180,E1 24745.071,E2 24745.071} C_VEL
LIN {X 0,Y 511.97,Z 628.679,A -85,B 0,C 180,E1 24742.795,E2 24742.795} C_VEL
LIN {X 0,Y 512.076,Z 622.622,A -85,B 0,C 180,E1 24740.561,E2 24740.561} C_VEL
LIN {X 0,Y 512.275,Z 615.097,A -85,B 0,C 180,E1 24738.403,E2 24738.403} C_VEL
LIN {X 0,Y 512.604,Z 605.712,A -85,B 0,C 180,E1 24736.234,E2 24736.234} C_VEL
LIN {X 0,Y 513.116,Z 594.186,A -85,B 0,C 180,E1 24734.054,E2 24734.054} C_VEL
LIN {X 0,Y 513.795,Z 580.955,A -85,B 0,C 180,E1 24731.977,E2 24731.977} C_VEL
LIN {X 0,Y 514.6,Z 566.862,A -85,B 0,C 180,E1 24730.119,E2 24730.119} C_VEL
LIN {X 0,Y 515.517,Z 551.771,A -85,B 0,C 180,E1 24728.43,E2 24728.43} C_VEL
LIN {X 0,Y 516.554,Z 535.043,A -85,B 0,C 180,E1 24726.842,E2 24726.842} C_VEL
LIN {X 0,Y 517.653,Z 516.946,A -85,B 0,C 180,E1 24725.403,E2 24725.403} C_VEL
LIN {X 0,Y 518.73,Z 498.286,A -85,B 0,C 180,E1 24724.176,E2 24724.176} C_VEL
LIN {X 0,Y 519.643,Z 480.565,A -85,B 0,C 180,E1 24723.226,E2 24723.226} C_VEL
LIN {X 0,Y 520.434,Z 460.214,A -85,B 0,C 180,E1 24722.385,E2 24722.385} C_VEL
LIN {X 0,Y 521.086,Z 439.918,A -85,B 0,C 180,E1 24721.76,E2 24721.76} C_VEL
LIN {X 0,Y 521.53,Z 418.981,A -85,B 0,C 180,E1 24721.317,E2 24721.317} C_VEL
LIN {X 0,Y 523.686,Z 192.289,A -85,B 0,C 180,E1 24717.978,E2 24717.978} C_VEL
LIN {X 0,Y 523.657,Z 176.59,A -85,B 0,C 180,E1 24717.728,E2 24717.728} C_VEL
LIN {X 0,Y 521.601,Z 163.135,A -85,B 0,C 180,E1 24717.377,E2 24717.377} C_VEL
LIN {X 0,Y 522.657,Z 131.203,A -85,B 0,C 180,E1 24715.154,E2 24715.154} C_VEL
LIN {X 0,Y 513.773,Z 108.921,A -85,B 0,C 180,E1 24712.838,E2 24712.838} C_VEL
LIN {X 0,Y 512.618,Z 105.633,A -85,B 0,C 180,E1 24712.481,E2 24712.481} C_VEL
LIN {X 0,Y 512.591,Z 105.631,A -85,B 0,C 180,E1 24709.185,E2 24709.185} C_VEL
LIN {X 0,Y 512.634,Z 105.627,A -85,B 0,C 180,E1 24705.87,E2 24705.87} C_VEL
LIN {X 0,Y 512.623,Z 105.626,A -85,B 0,C 180,E1 24702.443,E2 24702.443} C_VEL
LIN {X 0,Y 512.585,Z 105.608,A -85,B 0,C 180,E1 24699.074,E2 24699.074} C_VEL
LIN {X 0,Y 512.605,Z 105.633,A -85,B 0,C 180,E1 24695.677,E2 24695.677} C_VEL
LIN {X 0,Y 512.64,Z 105.622,A -85,B 0,C 180,E1 24692.304,E2 24692.304} C_VEL
LIN {X 0,Y 512.587,Z 105.626,A -85,B 0,C 180,E1 24689.058,E2 24689.058} C_VEL
LIN {X 0,Y 512.591,Z 105.63,A -85,B 0,C 180,E1 24685.536,E2 24685.536} C_VEL
LIN {X 0,Y 512.65,Z 105.626,A -85,B 0,C 180,E1 24682.233,E2 24682.233} C_VEL
LIN {X 0,Y 512.595,Z 105.623,A -85,B 0,C 180,E1 24678.892,E2 24678.892} C_VEL
LIN {X 0,Y 512.584,Z 105.631,A -85,B 0,C 180,E1 24675.5,E2 24675.5} C_VEL
LIN {X 0,Y 512.63,Z 105.623,A -85,B 0,C 180,E1 24672.16,E2 24672.16} C_VEL
LIN {X 0,Y 512.61,Z 105.63,A -85,B 0,C 180,E1 24668.751,E2 24668.751} C_VEL
LIN {X 0,Y 512.579,Z 105.63,A -85,B 0,C 180,E1 24665.372,E2 24665.372} C_VEL
LIN {X 0,Y 512.605,Z 105.622,A -85,B 0,C 180,E1 24662.012,E2 24662.012} C_VEL
LIN {X 0,Y 512.624,Z 105.627,A -85,B 0,C 180,E1 24658.659,E2 24658.659} C_VEL
LIN {X 0,Y 512.577,Z 105.624,A -85,B 0,C 180,E1 24655.3,E2 24655.3} C_VEL
LIN {X 0,Y 512.584,Z 105.633,A -85,B 0,C 180,E1 24651.813,E2 24651.813} C_VEL
LIN {X 0,Y 512.63,Z 105.62,A -85,B 0,C 180,E1 24648.41,E2 24648.41} C_VEL
LIN {X 0,Y 512.59,Z 105.632,A -85,B 0,C 180,E1 24645.079,E2 24645.079} C_VEL
LIN {X 0,Y 512.575,Z 105.626,A -85,B 0,C 180,E1 24641.696,E2 24641.696} C_VEL
LIN {X 0,Y 512.619,Z 105.627,A -85,B 0,C 180,E1 24638.368,E2 24638.368} C_VEL
LIN {X 0,Y 512.603,Z 105.628,A -85,B 0,C 180,E1 24634.959,E2 24634.959} C_VEL
LIN {X 0,Y 512.571,Z 105.621,A -85,B 0,C 180,E1 24631.578,E2 24631.578} C_VEL
LIN {X 0,Y 512.594,Z 105.629,A -85,B 0,C 180,E1 24628.22,E2 24628.22} C_VEL
LIN {X 0,Y 512.624,Z 105.632,A -85,B 0,C 180,E1 24624.808,E2 24624.808} C_VEL
LIN {X 0,Y 512.574,Z 105.632,A -85,B 0,C 180,E1 24621.462,E2 24621.462} C_VEL
LIN {X 0,Y 512.574,Z 105.634,A -85,B 0,C 180,E1 24618.003,E2 24618.003} C_VEL
LIN {X 0,Y 512.621,Z 105.634,A -85,B 0,C 180,E1 24614.6,E2 24614.6} C_VEL
LIN {X 0,Y 512.574,Z 105.635,A -85,B 0,C 180,E1 24614.034,E2 24614.034} C_VEL
LIN {X 0,Y 511.571,Z 105.761,A -85,B 0,C 180,E1 24613.173,E2 24613.173} C_VEL
LIN {X 0,Y 505.093,Z 106.568,A -85,B 0,C 180,E1 24610.69,E2 24610.69} C_VEL
LIN {X 0,Y 504.638,Z 106.621,A -85,B 0,C 180,E1 24610.122,E2 24610.122} C_VEL
LIN {X 0,Y 504.69,Z 106.622,A -85,B 0,C 180,E1 24606.833,E2 24606.833} C_VEL
LIN {X 0,Y 504.656,Z 106.751,A -85,B 0,C 180,E1 24604.12,E2 24604.12} C_VEL
LIN {X 0,Y 512.884,Z 130.022,A -85,B 0,C 180,E1 24601.235,E2 24601.235} C_VEL
LIN {X 0,Y 513.415,Z 132.758,A -85,B 0,C 180,E1 24600.938,E2 24600.938} C_VEL
LIN {X 0,Y 511.52,Z 172.113,A -85,B 0,C 180,E1 24597.448,E2 24597.448} C_VEL
LIN {X 0,Y 511.51,Z 174.889,A -85,B 0,C 180,E1 24597.238,E2 24597.238} C_VEL
LIN {X 0,Y 514.509,Z 191.733,A -85,B 0,C 180,E1 24596.793,E2 24596.793} C_VEL
LIN {X 0,Y 513.172,Z 387.492,A -85,B 0,C 180,E1 24594.037,E2 24594.037} C_VEL
LIN {X 0,Y 512.715,Z 406.444,A -85,B 0,C 180,E1 24593.556,E2 24593.556} C_VEL
LIN {X 0,Y 512.077,Z 423.554,A -85,B 0,C 180,E1 24592.925,E2 24592.925} C_VEL
LIN {X 0,Y 511.2,Z 441.169,A -85,B 0,C 180,E1 24592.056,E2 24592.056} C_VEL
LIN {X 0,Y 510.198,Z 457.671,A -85,B 0,C 180,E1 24591.015,E2 24591.015} C_VEL
LIN {X 0,Y 509.068,Z 473.886,A -85,B 0,C 180,E1 24589.743,E2 24589.743} C_VEL
LIN {X 0,Y 507.943,Z 488.931,A -85,B 0,C 180,E1 24588.298,E2 24588.298} C_VEL
LIN {X 0,Y 506.929,Z 502.396,A -85,B 0,C 180,E1 24586.735,E2 24586.735} C_VEL
LIN {X 0,Y 506.018,Z 514.818,A -85,B 0,C 180,E1 24585.001,E2 24585.001} C_VEL
LIN {X 0,Y 505.296,Z 525.767,A -85,B 0,C 180,E1 24583.152,E2 24583.152} C_VEL
LIN {X 0,Y 504.742,Z 535.293,A -85,B 0,C 180,E1 24581.193,E2 24581.193} C_VEL
LIN {X 0,Y 504.364,Z 543.332,A -85,B 0,C 180,E1 24579.124,E2 24579.124} C_VEL
LIN {X 0,Y 504.144,Z 549.816,A -85,B 0,C 180,E1 24576.948,E2 24576.948} C_VEL
LIN {X 0,Y 504.03,Z 554.436,A -85,B 0,C 180,E1 24574.778,E2 24574.778} C_VEL
LIN {X 0,Y 503.98,Z 557.31,A -85,B 0,C 180,E1 24572.615,E2 24572.615} C_VEL
LIN {X 0,Y 503.967,Z 558.513,A -85,B 0,C 180,E1 24570.454,E2 24570.454} C_VEL
LIN {X 0,Y 503.976,Z 558.07,A -85,B 0,C 180,E1 24568.294,E2 24568.294} C_VEL
LIN {X 0,Y 504.002,Z 555.972,A -85,B 0,C 180,E1 24566.132,E2 24566.132} C_VEL
LIN {X 0,Y 504.082,Z 552.164,A -85,B 0,C 180,E1 24563.965,E2 24563.965} C_VEL
LIN {X 0,Y 504.238,Z 546.894,A -85,B 0,C 180,E1 24561.906,E2 24561.906} C_VEL
LIN {X 0,Y 504.513,Z 539.883,A -85,B 0,C 180,E1 24559.84,E2 24559.84} C_VEL
LIN {X 0,Y 504.947,Z 531.469,A -85,B 0,C 180,E1 24557.883,E2 24557.883} C_VEL
LIN {X 0,Y 505.592,Z 521.058,A -85,B 0,C 180,E1 24555.921,E2 24555.921} C_VEL
LIN {X 0,Y 506.365,Z 509.897,A -85,B 0,C 180,E1 24554.187,E2 24554.187} C_VEL
LIN {X 0,Y 507.316,Z 497.165,A -85,B 0,C 180,E1 24552.537,E2 24552.537} C_VEL
LIN {X 0,Y 508.339,Z 483.503,A -85,B 0,C 180,E1 24551.062,E2 24551.062} C_VEL
LIN {X 0,Y 509.403,Z 468.952,A -85,B 0,C 180,E1 24549.756,E2 24549.756} C_VEL
LIN {X 0,Y 510.477,Z 452.904,A -85,B 0,C 180,E1 24548.574,E2 24548.574} C_VEL
LIN {X 0,Y 511.449,Z 436.222,A -85,B 0,C 180,E1 24547.59,E2 24547.59} C_VEL
LIN {X 0,Y 512.279,Z 418.416,A -85,B 0,C 180,E1 24546.779,E2 24546.779} C_VEL
LIN {X 0,Y 512.878,Z 399.988,A -85,B 0,C 180,E1 24546.169,E2 24546.169} C_VEL
LIN {X 0,Y 513.235,Z 381.239,A -85,B 0,C 180,E1 24545.766,E2 24545.766} C_VEL
LIN {X 0,Y 514.4,Z 189.94,A -85,B 0,C 180,E1 24543.081,E2 24543.081} C_VEL
LIN {X 0,Y 511.434,Z 174.262,A -85,B 0,C 180,E1 24542.649,E2 24542.649} C_VEL
LIN {X 0,Y 513.318,Z 135.111,A -85,B 0,C 180,E1 24539.184,E2 24539.184} C_VEL
LIN {X 0,Y 513.44,Z 131.636,A -85,B 0,C 180,E1 24538.866,E2 24538.866} C_VEL
LIN {X 0,Y 506.41,Z 111.849,A -85,B 0,C 180,E1 24536.429,E2 24536.429} C_VEL
LIN {X 0,Y 504.669,Z 106.624,A -85,B 0,C 180,E1 24535.759,E2 24535.759} C_VEL
LIN {X 0,Y 504.662,Z 106.618,A -85,B 0,C 180,E1 24532.394,E2 24532.394} C_VEL
LIN {X 0,Y 504.693,Z 106.619,A -85,B 0,C 180,E1 24529.009,E2 24529.009} C_VEL
LIN {X 0,Y 504.709,Z 106.618,A -85,B 0,C 180,E1 24525.468,E2 24525.468} C_VEL
LIN {X 0,Y 504.705,Z 106.619,A -85,B 0,C 180,E1 24521.884,E2 24521.884} C_VEL
LIN {X 0,Y 504.709,Z 106.62,A -85,B 0,C 180,E1 24518.322,E2 24518.322} C_VEL
LIN {X 0,Y 504.704,Z 106.619,A -85,B 0,C 180,E1 24514.789,E2 24514.789} C_VEL
LIN {X 0,Y 504.719,Z 106.696,A -85,B 0,C 180,E1 24513.108,E2 24513.108} C_VEL
LIN {X 0,Y 511.898,Z 128.896,A -85,B 0,C 180,E1 24510.781,E2 24510.781} C_VEL
LIN {X 0,Y 510.898,Z 168.767,A -85,B 0,C 180,E1 24507.508,E2 24507.508} C_VEL
LIN {X 0,Y 510.764,Z 179.564,A -85,B 0,C 180,E1 24506.653,E2 24506.653} C_VEL
LIN {X 0,Y 512.469,Z 191.432,A -85,B 0,C 180,E1 24506.363,E2 24506.363} C_VEL
LIN {X 0,Y 510.159,Z 388.809,A -85,B 0,C 180,E1 24503.278,E2 24503.278} C_VEL
LIN {X 0,Y 509.784,Z 408.012,A -85,B 0,C 180,E1 24502.767,E2 24502.767} C_VEL
LIN {X 0,Y 509.267,Z 426.137,A -85,B 0,C 180,E1 24502.074,E2 24502.074} C_VEL
LIN {X 0,Y 508.64,Z 443.415,A -85,B 0,C 180,E1 24501.205,E2 24501.205} C_VEL
LIN {X 0,Y 507.928,Z 460.473,A -85,B 0,C 180,E1 24500.118,E2 24500.118} C_VEL
LIN {X 0,Y 507.191,Z 476.451,A -85,B 0,C 180,E1 24498.863,E2 24498.863} C_VEL
LIN {X 0,Y 506.476,Z 491.142,A -85,B 0,C 180,E1 24497.462,E2 24497.462} C_VEL
LIN {X 0,Y 505.831,Z 504.35,A -85,B 0,C 180,E1 24495.948,E2 24495.948} C_VEL
LIN {X 0,Y 505.235,Z 516.945,A -85,B 0,C 180,E1 24494.205,E2 24494.205} C_VEL
LIN {X 0,Y 504.766,Z 527.941,A -85,B 0,C 180,E1 24492.353,E2 24492.353} C_VEL
LIN {X 0,Y 504.432,Z 536.858,A -85,B 0,C 180,E1 24490.507,E2 24490.507} C_VEL
LIN {X 0,Y 504.207,Z 544.398,A -85,B 0,C 180,E1 24488.553,E2 24488.553} C_VEL
LIN {X 0,Y 504.076,Z 550.486,A -85,B 0,C 180,E1 24486.492,E2 24486.492} C_VEL
LIN {X 0,Y 504,Z 554.804,A -85,B 0,C 180,E1 24484.438,E2 24484.438} C_VEL
LIN {X 0,Y 503.982,Z 557.472,A -85,B 0,C 180,E1 24482.388,E2 24482.388} C_VEL
LIN {X 0,Y 503.976,Z 558.571,A -85,B 0,C 180,E1 24480.341,E2 24480.341} C_VEL
LIN {X 0,Y 503.976,Z 558.126,A -85,B 0,C 180,E1 24478.295,E2 24478.295} C_VEL
LIN {X 0,Y 504.005,Z 555.976,A -85,B 0,C 180,E1 24476.133,E2 24476.133} C_VEL
LIN {X 0,Y 504.06,Z 552.279,A -85,B 0,C 180,E1 24474.08,E2 24474.08} C_VEL
LIN {X 0,Y 504.185,Z 546.858,A -85,B 0,C 180,E1 24472.021,E2 24472.021} C_VEL
LIN {X 0,Y 504.384,Z 539.995,A -85,B 0,C 180,E1 24470.069,E2 24470.069} C_VEL
LIN {X 0,Y 504.694,Z 531.403,A -85,B 0,C 180,E1 24468.147,E2 24468.147} C_VEL
LIN {X 0,Y 505.101,Z 521.598,A -85,B 0,C 180,E1 24466.375,E2 24466.375} C_VEL
LIN {X 0,Y 505.633,Z 509.871,A -85,B 0,C 180,E1 24464.635,E2 24464.635} C_VEL
LIN {X 0,Y 506.259,Z 496.512,A -85,B 0,C 180,E1 24463.005,E2 24463.005} C_VEL
LIN {X 0,Y 506.905,Z 482.349,A -85,B 0,C 180,E1 24461.58,E2 24461.58} C_VEL
LIN {X 0,Y 507.555,Z 467.086,A -85,B 0,C 180,E1 24460.314,E2 24460.314} C_VEL
LIN {X 0,Y 508.182,Z 450.427,A -85,B 0,C 180,E1 24459.192,E2 24459.192} C_VEL
LIN {X 0,Y 508.741,Z 432.897,A -85,B 0,C 180,E1 24458.256,E2 24458.256} C_VEL
LIN {X 0,Y 509.21,Z 413.957,A -85,B 0,C 180,E1 24457.487,E2 24457.487} C_VEL
LIN {X 0,Y 509.525,Z 395.209,A -85,B 0,C 180,E1 24456.947,E2 24456.947} C_VEL
LIN {X 0,Y 509.735,Z 372.875,A -85,B 0,C 180,E1 24456.55,E2 24456.55} C_VEL
LIN {X 0,Y 511.085,Z 255.585,A -85,B 0,C 180,E1 24454.709,E2 24454.709} C_VEL
LIN {X 0,Y 512.073,Z 188.827,A -85,B 0,C 180,E1 24453.563,E2 24453.563} C_VEL
LIN {X 0,Y 511.275,Z 183.477,A -85,B 0,C 180,E1 24453.395,E2 24453.395} C_VEL
LIN {X 0,Y 511.608,Z 147.45,A -85,B 0,C 180,E1 24450.624,E2 24450.624} C_VEL
LIN {X 0,Y 511.395,Z 126.269,A -85,B 0,C 180,E1 24449.02,E2 24449.02} C_VEL
LIN {X 0,Y 506.952,Z 112.722,A -85,B 0,C 180,E1 24447.691,E2 24447.691} C_VEL
LIN {X 0,Y 504.695,Z 106.622,A -85,B 0,C 180,E1 24447.057,E2 24447.057} C_VEL
LIN {X 0,Y 504.711,Z 106.62,A -85,B 0,C 180,E1 24443.536,E2 24443.536} C_VEL
LIN {X 0,Y 504.673,Z 106.622,A -85,B 0,C 180,E1 24440.061,E2 24440.061} C_VEL
LIN {X 0,Y 504.645,Z 106.623,A -85,B 0,C 180,E1 24436.648,E2 24436.648} C_VEL
LIN {X 0,Y 504.652,Z 106.623,A -85,B 0,C 180,E1 24433.188,E2 24433.188} C_VEL
LIN {X 0,Y 504.699,Z 106.621,A -85,B 0,C 180,E1 24429.766,E2 24429.766} C_VEL
LIN {X 0,Y 504.712,Z 106.846,A -85,B 0,C 180,E1 24428.051,E2 24428.051} C_VEL
LIN {X 0,Y 515.663,Z 134.499,A -85,B 0,C 180,E1 24425.103,E2 24425.103} C_VEL
LIN {X 0,Y 514.551,Z 163.973,A -85,B 0,C 180,E1 24423.049,E2 24423.049} C_VEL
LIN {X 0,Y 516.857,Z 180.462,A -85,B 0,C 180,E1 24422.635,E2 24422.635} C_VEL
LIN {X 0,Y 514.431,Z 400.86,A -85,B 0,C 180,E1 24419.32,E2 24419.32} C_VEL
LIN {X 0,Y 514.02,Z 428.87,A -85,B 0,C 180,E1 24418.855,E2 24418.855} C_VEL
LIN {X 0,Y 513.401,Z 449.53,A -85,B 0,C 180,E1 24418.313,E2 24418.313} C_VEL
LIN {X 0,Y 512.603,Z 470.016,A -85,B 0,C 180,E1 24417.567,E2 24417.567} C_VEL
LIN {X 0,Y 511.653,Z 490.621,A -85,B 0,C 180,E1 24416.584,E2 24416.584} C_VEL
LIN {X 0,Y 510.604,Z 509.544,A -85,B 0,C 180,E1 24415.457,E2 24415.457} C_VEL
LIN {X 0,Y 509.604,Z 526.843,A -85,B 0,C 180,E1 24414.21,E2 24414.21} C_VEL
LIN {X 0,Y 508.436,Z 544.203,A -85,B 0,C 180,E1 24412.672,E2 24412.672} C_VEL
LIN {X 0,Y 507.333,Z 560.418,A -85,B 0,C 180,E1 24410.96,E2 24410.96} C_VEL
LIN {X 0,Y 506.429,Z 574.208,A -85,B 0,C 180,E1 24409.252,E2 24409.252} C_VEL
LIN {X 0,Y 505.606,Z 587.865,A -85,B 0,C 180,E1 24407.256,E2 24407.256} C_VEL
LIN {X 0,Y 504.957,Z 599.912,A -85,B 0,C 180,E1 24405.152,E2 24405.152} C_VEL
LIN {X 0,Y 504.502,Z 609.872,A -85,B 0,C 180,E1 24403.058,E2 24403.058} C_VEL
LIN {X 0,Y 504.206,Z 618.462,A -85,B 0,C 180,E1 24400.859,E2 24400.859} C_VEL
LIN {X 0,Y 504.026,Z 625.592,A -85,B 0,C 180,E1 24398.557,E2 24398.557} C_VEL
LIN {X 0,Y 503.941,Z 630.725,A -85,B 0,C 180,E1 24396.38,E2 24396.38} C_VEL
LIN {X 0,Y 503.915,Z 634.403,A -85,B 0,C 180,E1 24394.097,E2 24394.097} C_VEL
LIN {X 0,Y 503.908,Z 636.44,A -85,B 0,C 180,E1 24391.82,E2 24391.82} C_VEL
LIN {X 0,Y 503.9,Z 636.895,A -85,B 0,C 180,E1 24389.432,E2 24389.432} C_VEL
LIN {X 0,Y 503.914,Z 635.732,A -85,B 0,C 180,E1 24387.157,E2 24387.157} C_VEL
LIN {X 0,Y 503.927,Z 632.969,A -85,B 0,C 180,E1 24384.878,E2 24384.878} C_VEL
LIN {X 0,Y 503.978,Z 628.483,A -85,B 0,C 180,E1 24382.592,E2 24382.592} C_VEL
LIN {X 0,Y 504.104,Z 622.268,A -85,B 0,C 180,E1 24380.295,E2 24380.295} C_VEL
LIN {X 0,Y 504.339,Z 614.179,A -85,B 0,C 180,E1 24377.986,E2 24377.986} C_VEL
LIN {X 0,Y 504.73,Z 604.564,A -85,B 0,C 180,E1 24375.781,E2 24375.781} C_VEL
LIN {X 0,Y 505.289,Z 593.48,A -85,B 0,C 180,E1 24373.68,E2 24373.68} C_VEL
LIN {X 0,Y 506.015,Z 580.957,A -85,B 0,C 180,E1 24371.69,E2 24371.69} C_VEL
LIN {X 0,Y 506.904,Z 566.893,A -85,B 0,C 180,E1 24369.808,E2 24369.808} C_VEL
LIN {X 0,Y 507.914,Z 551.839,A -85,B 0,C 180,E1 24368.098,E2 24368.098} C_VEL
LIN {X 0,Y 509.048,Z 535.284,A -85,B 0,C 180,E1 24366.502,E2 24366.502} C_VEL
LIN {X 0,Y 510.028,Z 519.897,A -85,B 0,C 180,E1 24365.258,E2 24365.258} C_VEL
LIN {X 0,Y 511.089,Z 501.109,A -85,B 0,C 180,E1 24364.011,E2 24364.011} C_VEL
LIN {X 0,Y 512.135,Z 480.554,A -85,B 0,C 180,E1 24362.906,E2 24362.906} C_VEL
LIN {X 0,Y 512.996,Z 460.168,A -85,B 0,C 180,E1 24362.048,E2 24362.048} C_VEL
LIN {X 0,Y 513.713,Z 440.035,A -85,B 0,C 180,E1 24361.414,E2 24361.414} C_VEL
LIN {X 0,Y 514.219,Z 418.828,A -85,B 0,C 180,E1 24360.954,E2 24360.954} C_VEL
LIN {X 0,Y 516.679,Z 193.943,A -85,B 0,C 180,E1 24357.571,E2 24357.571} C_VEL
LIN {X 0,Y 516.656,Z 177.718,A -85,B 0,C 180,E1 24357.308,E2 24357.308} C_VEL
LIN {X 0,Y 514.49,Z 162.907,A -85,B 0,C 180,E1 24356.902,E2 24356.902} C_VEL
LIN {X 0,Y 515.574,Z 134.277,A -85,B 0,C 180,E1 24354.875,E2 24354.875} C_VEL
LIN {X 0,Y 506.973,Z 112.783,A -85,B 0,C 180,E1 24352.596,E2 24352.596} C_VEL
LIN {X 0,Y 504.703,Z 106.617,A -85,B 0,C 180,E1 24351.896,E2 24351.896} C_VEL
LIN {X 0,Y 504.679,Z 106.615,A -85,B 0,C 180,E1 24348.494,E2 24348.494} C_VEL
LIN {X 0,Y 504.651,Z 106.622,A -85,B 0,C 180,E1 24345.145,E2 24345.145} C_VEL
LIN {X 0,Y 504.672,Z 106.621,A -85,B 0,C 180,E1 24341.678,E2 24341.678} C_VEL
LIN {X 0,Y 504.696,Z 106.586,A -85,B 0,C 180,E1 24338.322,E2 24338.322} C_VEL
LIN {X 0,Y 504.655,Z 106.62,A -85,B 0,C 180,E1 24334.892,E2 24334.892} C_VEL
LIN {X 0,Y 504.65,Z 106.621,A -85,B 0,C 180,E1 24331.36,E2 24331.36} C_VEL
LIN {X 0,Y 504.691,Z 106.614,A -85,B 0,C 180,E1 24328.003,E2 24328.003} C_VEL
LIN {X 0,Y 504.68,Z 106.616,A -85,B 0,C 180,E1 24324.585,E2 24324.585} C_VEL
LIN {X 0,Y 504.646,Z 106.62,A -85,B 0,C 180,E1 24321.258,E2 24321.258} C_VEL
LIN {X 0,Y 504.66,Z 106.619,A -85,B 0,C 180,E1 24317.765,E2 24317.765} C_VEL
LIN {X 0,Y 504.711,Z 106.611,A -85,B 0,C 180,E1 24314.337,E2 24314.337} C_VEL
LIN {X 0,Y 504.661,Z 106.618,A -85,B 0,C 180,E1 24310.849,E2 24310.849} C_VEL
LIN {X 0,Y 504.639,Z 106.608,A -85,B 0,C 180,E1 24307.399,E2 24307.399} C_VEL
LIN {X 0,Y 504.665,Z 106.621,A -85,B 0,C 180,E1 24303.976,E2 24303.976} C_VEL
LIN {X 0,Y 504.694,Z 106.605,A -85,B 0,C 180,E1 24300.567,E2 24300.567} C_VEL
LIN {X 0,Y 504.646,Z 106.621,A -85,B 0,C 180,E1 24297.161,E2 24297.161} C_VEL
LIN {X 0,Y 504.638,Z 106.616,A -85,B 0,C 180,E1 24293.629,E2 24293.629} C_VEL
LIN {X 0,Y 504.684,Z 106.616,A -85,B 0,C 180,E1 24290.305,E2 24290.305} C_VEL
LIN {X 0,Y 504.672,Z 106.614,A -85,B 0,C 180,E1 24286.83,E2 24286.83} C_VEL
LIN {X 0,Y 504.635,Z 106.616,A -85,B 0,C 180,E1 24283.527,E2 24283.527} C_VEL
LIN {X 0,Y 504.654,Z 106.622,A -85,B 0,C 180,E1 24280.075,E2 24280.075} C_VEL
LIN {X 0,Y 504.695,Z 106.608,A -85,B 0,C 180,E1 24276.657,E2 24276.657} C_VEL
LIN {X 0,Y 504.643,Z 106.62,A -85,B 0,C 180,E1 24273.271,E2 24273.271} C_VEL
LIN {X 0,Y 504.633,Z 106.621,A -85,B 0,C 180,E1 24269.752,E2 24269.752} C_VEL
LIN {X 0,Y 504.675,Z 106.615,A -85,B 0,C 180,E1 24266.444,E2 24266.444} C_VEL
LIN {X 0,Y 504.67,Z 106.617,A -85,B 0,C 180,E1 24262.966,E2 24262.966} C_VEL
LIN {X 0,Y 504.631,Z 106.621,A -85,B 0,C 180,E1 24259.616,E2 24259.616} C_VEL
LIN {X 0,Y 504.638,Z 106.617,A -85,B 0,C 180,E1 24256.094,E2 24256.094} C_VEL
LIN {X 0,Y 504.684,Z 106.617,A -85,B 0,C 180,E1 24252.652,E2 24252.652} C_VEL
LIN {X 0,Y 504.638,Z 106.621,A -85,B 0,C 180,E1 24250.122,E2 24250.122} C_VEL
LIN {X 0,Y 503.629,Z 106.751,A -85,B 0,C 180,E1 24249.248,E2 24249.248} C_VEL
LIN {X 0,Y 497.152,Z 107.562,A -85,B 0,C 180,E1 24246.725,E2 24246.725} C_VEL
LIN {X 0,Y 496.7,Z 107.612,A -85,B 0,C 180,E1 24246.148,E2 24246.148} C_VEL
LIN {X 0,Y 496.768,Z 107.773,A -85,B 0,C 180,E1 24244.683,E2 24244.683} C_VEL
LIN {X 0,Y 505.204,Z 131.415,A -85,B 0,C 180,E1 24241.677,E2 24241.677} C_VEL
LIN {X 0,Y 506.244,Z 135.388,A -85,B 0,C 180,E1 24241.218,E2 24241.218} C_VEL
LIN {X 0,Y 504.222,Z 174.283,A -85,B 0,C 180,E1 24237.73,E2 24237.73} C_VEL
LIN {X 0,Y 507.555,Z 193.03,A -85,B 0,C 180,E1 24237.223,E2 24237.223} C_VEL
LIN {X 0,Y 506.096,Z 387.988,A -85,B 0,C 180,E1 24234.453,E2 24234.453} C_VEL
LIN {X 0,Y 505.616,Z 406.86,A -85,B 0,C 180,E1 24233.97,E2 24233.97} C_VEL
LIN {X 0,Y 504.937,Z 424.111,A -85,B 0,C 180,E1 24233.329,E2 24233.329} C_VEL
LIN {X 0,Y 504.003,Z 441.809,A -85,B 0,C 180,E1 24232.45,E2 24232.45} C_VEL
LIN {X 0,Y 502.937,Z 458.419,A -85,B 0,C 180,E1 24231.395,E2 24231.395} C_VEL
LIN {X 0,Y 501.726,Z 474.705,A -85,B 0,C 180,E1 24230.105,E2 24230.105} C_VEL
LIN {X 0,Y 500.551,Z 489.234,A -85,B 0,C 180,E1 24228.698,E2 24228.698} C_VEL
LIN {X 0,Y 499.429,Z 502.745,A -85,B 0,C 180,E1 24227.114,E2 24227.114} C_VEL
LIN {X 0,Y 498.403,Z 515.194,A -85,B 0,C 180,E1 24225.355,E2 24225.355} C_VEL
LIN {X 0,Y 497.561,Z 526.361,A -85,B 0,C 180,E1 24223.441,E2 24223.441} C_VEL
LIN {X 0,Y 496.938,Z 535.691,A -85,B 0,C 180,E1 24221.489,E2 24221.489} C_VEL
LIN {X 0,Y 496.494,Z 543.743,A -85,B 0,C 180,E1 24219.387,E2 24219.387} C_VEL
LIN {X 0,Y 496.231,Z 549.971,A -85,B 0,C 180,E1 24217.292,E2 24217.292} C_VEL
LIN {X 0,Y 496.081,Z 554.732,A -85,B 0,C 180,E1 24215.087,E2 24215.087} C_VEL
LIN {X 0,Y 496.015,Z 557.754,A -85,B 0,C 180,E1 24212.888,E2 24212.888} C_VEL
LIN {X 0,Y 496,Z 559.116,A -85,B 0,C 180,E1 24210.692,E2 24210.692} C_VEL
LIN {X 0,Y 496.002,Z 558.849,A -85,B 0,C 180,E1 24208.498,E2 24208.498} C_VEL
LIN {X 0,Y 496.03,Z 556.947,A -85,B 0,C 180,E1 24206.301,E2 24206.301} C_VEL
LIN {X 0,Y 496.122,Z 553.359,A -85,B 0,C 180,E1 24204.1,E2 24204.1} C_VEL
LIN {X 0,Y 496.309,Z 547.993,A -85,B 0,C 180,E1 24201.892,E2 24201.892} C_VEL
LIN {X 0,Y 496.644,Z 540.715,A -85,B 0,C 180,E1 24199.677,E2 24199.677} C_VEL
LIN {X 0,Y 497.142,Z 532.39,A -85,B 0,C 180,E1 24197.69,E2 24197.69} C_VEL
LIN {X 0,Y 497.867,Z 522.094,A -85,B 0,C 180,E1 24195.698,E2 24195.698} C_VEL
LIN {X 0,Y 498.729,Z 511.052,A -85,B 0,C 180,E1 24193.938,E2 24193.938} C_VEL
LIN {X 0,Y 499.809,Z 498.08,A -85,B 0,C 180,E1 24192.22,E2 24192.22} C_VEL
LIN {X 0,Y 500.94,Z 484.388,A -85,B 0,C 180,E1 24190.716,E2 24190.716} C_VEL
LIN {X 0,Y 502.118,Z 469.438,A -85,B 0,C 180,E1 24189.362,E2 24189.362} C_VEL
LIN {X 0,Y 503.239,Z 453.603,A -85,B 0,C 180,E1 24188.189,E2 24188.189} C_VEL
LIN {X 0,Y 504.264,Z 436.922,A -85,B 0,C 180,E1 24187.198,E2 24187.198} C_VEL
LIN {X 0,Y 505.118,Z 419.717,A -85,B 0,C 180,E1 24186.403,E2 24186.403} C_VEL
LIN {X 0,Y 505.775,Z 400.89,A -85,B 0,C 180,E1 24185.766,E2 24185.766} C_VEL
LIN {X 0,Y 506.166,Z 381.858,A -85,B 0,C 180,E1 24185.351,E2 24185.351} C_VEL
LIN {X 0,Y 507.446,Z 191.24,A -85,B 0,C 180,E1 24182.65,E2 24182.65} C_VEL
LIN {X 0,Y 504.23,Z 174.239,A -85,B 0,C 180,E1 24182.177,E2 24182.177} C_VEL
LIN {X 0,Y 506.284,Z 134.784,A -85,B 0,C 180,E1 24178.635,E2 24178.635} C_VEL
LIN {X 0,Y 499.595,Z 115.776,A -85,B 0,C 180,E1 24176.259,E2 24176.259} C_VEL
LIN {X 0,Y 496.76,Z 107.611,A -85,B 0,C 180,E1 24175.174,E2 24175.174} C_VEL
LIN {X 0,Y 496.756,Z 107.586,A -85,B 0,C 180,E1 24171.688,E2 24171.688} C_VEL
LIN {X 0,Y 496.743,Z 107.612,A -85,B 0,C 180,E1 24168.221,E2 24168.221} C_VEL
LIN {X 0,Y 496.746,Z 107.609,A -85,B 0,C 180,E1 24164.626,E2 24164.626} C_VEL
LIN {X 0,Y 496.767,Z 107.603,A -85,B 0,C 180,E1 24161.16,E2 24161.16} C_VEL
LIN {X 0,Y 496.76,Z 107.604,A -85,B 0,C 180,E1 24157.58,E2 24157.58} C_VEL
LIN {X 0,Y 496.75,Z 107.61,A -85,B 0,C 180,E1 24153.975,E2 24153.975} C_VEL
LIN {X 0,Y 496.764,Z 107.654,A -85,B 0,C 180,E1 24153.562,E2 24153.562} C_VEL
LIN {X 0,Y 504.574,Z 131.223,A -85,B 0,C 180,E1 24151.049,E2 24151.049} C_VEL
LIN {X 0,Y 503.545,Z 170.356,A -85,B 0,C 180,E1 24147.816,E2 24147.816} C_VEL
LIN {X 0,Y 503.419,Z 180.042,A -85,B 0,C 180,E1 24147.049,E2 24147.049} C_VEL
LIN {X 0,Y 505.229,Z 192.587,A -85,B 0,C 180,E1 24146.734,E2 24146.734} C_VEL
LIN {X 0,Y 502.677,Z 389.302,A -85,B 0,C 180,E1 24143.593,E2 24143.593} C_VEL
LIN {X 0,Y 502.274,Z 408.518,A -85,B 0,C 180,E1 24143.074,E2 24143.074} C_VEL
LIN {X 0,Y 501.722,Z 426.592,A -85,B 0,C 180,E1 24142.373,E2 24142.373} C_VEL
LIN {X 0,Y 501.043,Z 444.069,A -85,B 0,C 180,E1 24141.481,E2 24141.481} C_VEL
LIN {X 0,Y 500.288,Z 460.942,A -85,B 0,C 180,E1 24140.391,E2 24140.391} C_VEL
LIN {X 0,Y 499.501,Z 476.884,A -85,B 0,C 180,E1 24139.123,E2 24139.123} C_VEL
LIN {X 0,Y 498.722,Z 491.79,A -85,B 0,C 180,E1 24137.682,E2 24137.682} C_VEL
LIN {X 0,Y 498.002,Z 505.47,A -85,B 0,C 180,E1 24136.086,E2 24136.086} C_VEL
LIN {X 0,Y 497.363,Z 518.058,A -85,B 0,C 180,E1 24134.308,E2 24134.308} C_VEL
LIN {X 0,Y 496.862,Z 528.953,A -85,B 0,C 180,E1 24132.435,E2 24132.435} C_VEL
LIN {X 0,Y 496.503,Z 537.821,A -85,B 0,C 180,E1 24130.56,E2 24130.56} C_VEL
LIN {X 0,Y 496.258,Z 545.312,A -85,B 0,C 180,E1 24128.575,E2 24128.575} C_VEL
LIN {X 0,Y 496.115,Z 551.352,A -85,B 0,C 180,E1 24126.481,E2 24126.481} C_VEL
LIN {X 0,Y 496.031,Z 555.617,A -85,B 0,C 180,E1 24124.393,E2 24124.393} C_VEL
LIN {X 0,Y 496.009,Z 558.341,A -85,B 0,C 180,E1 24122.195,E2 24122.195} C_VEL
LIN {X 0,Y 496.006,Z 559.309,A -85,B 0,C 180,E1 24120,E2 24120} C_VEL
LIN {X 0,Y 496.013,Z 558.531,A -85,B 0,C 180,E1 24117.805,E2 24117.805} C_VEL
LIN {X 0,Y 496.048,Z 555.984,A -85,B 0,C 180,E1 24115.607,E2 24115.607} C_VEL
LIN {X 0,Y 496.14,Z 551.795,A -85,B 0,C 180,E1 24113.482,E2 24113.482} C_VEL
LIN {X 0,Y 496.288,Z 546.013,A -85,B 0,C 180,E1 24111.426,E2 24111.426} C_VEL
LIN {X 0,Y 496.542,Z 538.664,A -85,B 0,C 180,E1 24109.442,E2 24109.442} C_VEL
LIN {X 0,Y 496.905,Z 529.917,A -85,B 0,C 180,E1 24107.567,E2 24107.567} C_VEL
LIN {X 0,Y 497.367,Z 519.813,A -85,B 0,C 180,E1 24105.803,E2 24105.803} C_VEL
LIN {X 0,Y 497.94,Z 508.129,A -85,B 0,C 180,E1 24104.12,E2 24104.12} C_VEL
LIN {X 0,Y 498.621,Z 494.471,A -85,B 0,C 180,E1 24102.495,E2 24102.495} C_VEL
LIN {X 0,Y 499.353,Z 479.273,A -85,B 0,C 180,E1 24101.012,E2 24101.012} C_VEL
LIN {X 0,Y 500.05,Z 463.604,A -85,B 0,C 180,E1 24099.763,E2 24099.763} C_VEL
LIN {X 0,Y 500.707,Z 447.043,A -85,B 0,C 180,E1 24098.689,E2 24098.689} C_VEL
LIN {X 0,Y 501.274,Z 429.553,A -85,B 0,C 180,E1 24097.791,E2 24097.791} C_VEL
LIN {X 0,Y 501.73,Z 410.834,A -85,B 0,C 180,E1 24097.069,E2 24097.069} C_VEL
LIN {X 0,Y 502.03,Z 391.743,A -85,B 0,C 180,E1 24096.562,E2 24096.562} C_VEL
LIN {X 0,Y 503.879,Z 251.277,A -85,B 0,C 180,E1 24094.26,E2 24094.26} C_VEL
LIN {X 0,Y 504.96,Z 190.01,A -85,B 0,C 180,E1 24093.163,E2 24093.163} C_VEL
LIN {X 0,Y 504.15,Z 184.62,A -85,B 0,C 180,E1 24092.989,E2 24092.989} C_VEL
LIN {X 0,Y 504.565,Z 146.477,A -85,B 0,C 180,E1 24090.042,E2 24090.042} C_VEL
LIN {X 0,Y 504.362,Z 129.102,A -85,B 0,C 180,E1 24088.709,E2 24088.709} C_VEL
LIN {X 0,Y 499.881,Z 115.745,A -85,B 0,C 180,E1 24087.361,E2 24087.361} C_VEL
LIN {X 0,Y 496.728,Z 107.612,A -85,B 0,C 180,E1 24086.485,E2 24086.485} C_VEL
LIN {X 0,Y 496.738,Z 107.613,A -85,B 0,C 180,E1 24082.998,E2 24082.998} C_VEL
LIN {X 0,Y 496.772,Z 107.608,A -85,B 0,C 180,E1 24079.536,E2 24079.536} C_VEL
LIN {X 0,Y 496.737,Z 107.612,A -85,B 0,C 180,E1 24076.018,E2 24076.018} C_VEL
LIN {X 0,Y 496.7,Z 107.613,A -85,B 0,C 180,E1 24072.561,E2 24072.561} C_VEL
LIN {X 0,Y 496.7,Z 107.615,A -85,B 0,C 180,E1 24069.012,E2 24069.012} C_VEL
LIN {X 0,Y 496.725,Z 107.796,A -85,B 0,C 180,E1 24068.648,E2 24068.648} C_VEL
LIN {X 0,Y 506.744,Z 132.944,A -85,B 0,C 180,E1 24065.875,E2 24065.875} C_VEL
LIN {X 0,Y 508.562,Z 138.19,A -85,B 0,C 180,E1 24065.343,E2 24065.343} C_VEL
LIN {X 0,Y 507.461,Z 164.094,A -85,B 0,C 180,E1 24063.513,E2 24063.513} C_VEL
LIN {X 0,Y 509.898,Z 181.695,A -85,B 0,C 180,E1 24063.062,E2 24063.062} C_VEL
LIN {X 0,Y 507.195,Z 398.406,A -85,B 0,C 180,E1 24059.735,E2 24059.735} C_VEL
LIN {X 0,Y 506.727,Z 428.104,A -85,B 0,C 180,E1 24059.238,E2 24059.238} C_VEL
LIN {X 0,Y 506.047,Z 448.694,A -85,B 0,C 180,E1 24058.694,E2 24058.694} C_VEL
LIN {X 0,Y 505.234,Z 468.439,A -85,B 0,C 180,E1 24057.972,E2 24057.972} C_VEL
LIN {X 0,Y 504.211,Z 488.624,A -85,B 0,C 180,E1 24057.008,E2 24057.008} C_VEL
LIN {X 0,Y 503.137,Z 506.895,A -85,B 0,C 180,E1 24055.926,E2 24055.926} C_VEL
LIN {X 0,Y 502.018,Z 525.407,A -85,B 0,C 180,E1 24054.599,E2 24054.599} C_VEL
LIN {X 0,Y 500.867,Z 542.953,A -85,B 0,C 180,E1 24053.096,E2 24053.096} C_VEL
LIN {X 0,Y 499.849,Z 558.295,A -85,B 0,C 180,E1 24051.543,E2 24051.543} C_VEL
LIN {X 0,Y 498.835,Z 572.436,A -85,B 0,C 180,E1 24049.801,E2 24049.801} C_VEL
LIN {X 0,Y 497.919,Z 585.802,A -85,B 0,C 180,E1 24047.857,E2 24047.857} C_VEL
LIN {X 0,Y 497.218,Z 597.37,A -85,B 0,C 180,E1 24045.872,E2 24045.872} C_VEL
LIN {X 0,Y 496.651,Z 608.328,A -85,B 0,C 180,E1 24043.624,E2 24043.624} C_VEL
LIN {X 0,Y 496.291,Z 617.247,A -85,B 0,C 180,E1 24041.388,E2 24041.388} C_VEL
LIN {X 0,Y 496.082,Z 624.372,A -85,B 0,C 180,E1 24039.163,E2 24039.163} C_VEL
LIN {X 0,Y 495.968,Z 630.004,A -85,B 0,C 180,E1 24036.832,E2 24036.832} C_VEL
LIN {X 0,Y 495.913,Z 633.926,A -85,B 0,C 180,E1 24034.511,E2 24034.511} C_VEL
LIN {X 0,Y 495.908,Z 636.304,A -85,B 0,C 180,E1 24032.081,E2 24032.081} C_VEL
LIN {X 0,Y 495.906,Z 636.962,A -85,B 0,C 180,E1 24029.77,E2 24029.77} C_VEL
LIN {X 0,Y 495.904,Z 636.031,A -85,B 0,C 180,E1 24027.458,E2 24027.458} C_VEL
LIN {X 0,Y 495.926,Z 633.448,A -85,B 0,C 180,E1 24025.143,E2 24025.143} C_VEL
LIN {X 0,Y 495.978,Z 629.246,A -85,B 0,C 180,E1 24022.821,E2 24022.821} C_VEL
LIN {X 0,Y 496.102,Z 623.328,A -85,B 0,C 180,E1 24020.488,E2 24020.488} C_VEL
LIN {X 0,Y 496.34,Z 615.946,A -85,B 0,C 180,E1 24018.245,E2 24018.245} C_VEL
LIN {X 0,Y 496.736,Z 606.583,A -85,B 0,C 180,E1 24015.976,E2 24015.976} C_VEL
LIN {X 0,Y 497.293,Z 596.109,A -85,B 0,C 180,E1 24013.892,E2 24013.892} C_VEL
LIN {X 0,Y 498.034,Z 584.042,A -85,B 0,C 180,E1 24011.871,E2 24011.871} C_VEL
LIN {X 0,Y 499.023,Z 569.67,A -85,B 0,C 180,E1 24009.842,E2 24009.842} C_VEL
LIN {X 0,Y 500.037,Z 555.622,A -85,B 0,C 180,E1 24008.167,E2 24008.167} C_VEL
LIN {X 0,Y 501.127,Z 539.112,A -85,B 0,C 180,E1 24006.545,E2 24006.545} C_VEL
LIN {X 0,Y 502.316,Z 520.821,A -85,B 0,C 180,E1 24005.041,E2 24005.041} C_VEL
LIN {X 0,Y 503.437,Z 502.23,A -85,B 0,C 180,E1 24003.776,E2 24003.776} C_VEL
LIN {X 0,Y 504.51,Z 482.77,A -85,B 0,C 180,E1 24002.692,E2 24002.692} C_VEL
LIN {X 0,Y 505.45,Z 463.109,A -85,B 0,C 180,E1 24001.818,E2 24001.818} C_VEL
LIN {X 0,Y 506.301,Z 441.722,A -85,B 0,C 180,E1 24001.101,E2 24001.101} C_VEL
LIN {X 0,Y 506.887,Z 420.739,A -85,B 0,C 180,E1 24000.616,E2 24000.616} C_VEL
LIN {X 0,Y 509.679,Z 196.081,A -85,B 0,C 180,E1 23997.163,E2 23997.163} C_VEL
LIN {X 0,Y 509.714,Z 178.996,A -85,B 0,C 180,E1 23996.881,E2 23996.881} C_VEL
LIN {X 0,Y 507.394,Z 163.13,A -85,B 0,C 180,E1 23996.445,E2 23996.445} C_VEL
LIN {X 0,Y 508.499,Z 137.363,A -85,B 0,C 180,E1 23994.59,E2 23994.59} C_VEL
LIN {X 0,Y 499.194,Z 113.971,A -85,B 0,C 180,E1 23992.056,E2 23992.056} C_VEL
LIN {X 0,Y 496.719,Z 107.61,A -85,B 0,C 180,E1 23991.318,E2 23991.318} C_VEL
LIN {X 0,Y 496.756,Z 107.603,A -85,B 0,C 180,E1 23987.915,E2 23987.915} C_VEL
LIN {X 0,Y 496.752,Z 107.609,A -85,B 0,C 180,E1 23984.396,E2 23984.396} C_VEL
LIN {X 0,Y 496.714,Z 107.608,A -85,B 0,C 180,E1 23980.989,E2 23980.989} C_VEL
LIN {X 0,Y 496.714,Z 107.588,A -85,B 0,C 180,E1 23977.438,E2 23977.438} C_VEL
LIN {X 0,Y 496.753,Z 107.603,A -85,B 0,C 180,E1 23973.978,E2 23973.978} C_VEL
LIN {X 0,Y 496.751,Z 107.608,A -85,B 0,C 180,E1 23970.479,E2 23970.479} C_VEL
LIN {X 0,Y 496.711,Z 107.608,A -85,B 0,C 180,E1 23967.06,E2 23967.06} C_VEL
LIN {X 0,Y 496.711,Z 107.604,A -85,B 0,C 180,E1 23963.488,E2 23963.488} C_VEL
LIN {X 0,Y 496.756,Z 107.602,A -85,B 0,C 180,E1 23960.132,E2 23960.132} C_VEL
LIN {X 0,Y 496.744,Z 107.606,A -85,B 0,C 180,E1 23956.608,E2 23956.608} C_VEL
LIN {X 0,Y 496.704,Z 107.596,A -85,B 0,C 180,E1 23953.266,E2 23953.266} C_VEL
LIN {X 0,Y 496.715,Z 107.609,A -85,B 0,C 180,E1 23949.735,E2 23949.735} C_VEL
LIN {X 0,Y 496.765,Z 107.594,A -85,B 0,C 180,E1 23946.355,E2 23946.355} C_VEL
LIN {X 0,Y 496.723,Z 107.609,A -85,B 0,C 180,E1 23942.884,E2 23942.884} C_VEL
LIN {X 0,Y 496.701,Z 107.606,A -85,B 0,C 180,E1 23939.423,E2 23939.423} C_VEL
LIN {X 0,Y 496.716,Z 107.602,A -85,B 0,C 180,E1 23935.96,E2 23935.96} C_VEL
LIN {X 0,Y 496.767,Z 107.604,A -85,B 0,C 180,E1 23932.482,E2 23932.482} C_VEL
LIN {X 0,Y 496.719,Z 107.603,A -85,B 0,C 180,E1 23928.975,E2 23928.975} C_VEL
LIN {X 0,Y 496.699,Z 107.611,A -85,B 0,C 180,E1 23925.521,E2 23925.521} C_VEL
LIN {X 0,Y 496.716,Z 107.601,A -85,B 0,C 180,E1 23922.062,E2 23922.062} C_VEL
LIN {X 0,Y 496.759,Z 107.607,A -85,B 0,C 180,E1 23918.635,E2 23918.635} C_VEL
LIN {X 0,Y 496.707,Z 107.605,A -85,B 0,C 180,E1 23915.208,E2 23915.208} C_VEL
LIN {X 0,Y 496.695,Z 107.598,A -85,B 0,C 180,E1 23911.767,E2 23911.767} C_VEL
LIN {X 0,Y 496.731,Z 107.606,A -85,B 0,C 180,E1 23908.367,E2 23908.367} C_VEL
LIN {X 0,Y 496.742,Z 107.609,A -85,B 0,C 180,E1 23904.853,E2 23904.853} C_VEL
LIN {X 0,Y 496.7,Z 107.61,A -85,B 0,C 180,E1 23901.389,E2 23901.389} C_VEL
LIN {X 0,Y 496.694,Z 107.612,A -85,B 0,C 180,E1 23897.906,E2 23897.906} C_VEL
LIN {X 0,Y 496.727,Z 107.613,A -85,B 0,C 180,E1 23894.465,E2 23894.465} C_VEL
LIN {X 0,Y 496.737,Z 107.612,A -85,B 0,C 180,E1 23890.99,E2 23890.99} C_VEL
LIN {X 0,Y 496.695,Z 107.61,A -85,B 0,C 180,E1 23887.584,E2 23887.584} C_VEL
LIN {X 0,Y 496.7,Z 107.612,A -85,B 0,C 180,E1 23886.148,E2 23886.148} C_VEL
LIN {X 0,Y 496.434,Z 108.527,A -85,B 0,C 180,E1 23885.53,E2 23885.53} C_VEL
LIN {X 0,Y 495.758,Z 111.407,A -85,B 0,C 180,E1 23884.846,E2 23884.846} C_VEL
LIN {X 0,Y 494.877,Z 117.064,A -85,B 0,C 180,E1 23884.033,E2 23884.033} C_VEL
LIN {X 0,Y 494.908,Z 124.465,A -85,B 0,C 180,E1 23883.175,E2 23883.175} C_VEL
LIN {X 0,Y 495.655,Z 127.638,A -85,B 0,C 180,E1 23882.793,E2 23882.793} C_VEL
LIN {X 0,Y 499.096,Z 137.824,A -85,B 0,C 180,E1 23881.524,E2 23881.524} C_VEL
LIN {X 0,Y 497.099,Z 174.442,A -85,B 0,C 180,E1 23878.215,E2 23878.215} C_VEL
LIN {X 0,Y 500.63,Z 194.311,A -85,B 0,C 180,E1 23877.665,E2 23877.665} C_VEL
LIN {X 0,Y 499.027,Z 388.367,A -85,B 0,C 180,E1 23874.878,E2 23874.878} C_VEL
LIN {X 0,Y 498.512,Z 407.344,A -85,B 0,C 180,E1 23874.387,E2 23874.387} C_VEL
LIN {X 0,Y 497.724,Z 425.735,A -85,B 0,C 180,E1 23873.688,E2 23873.688} C_VEL
LIN {X 0,Y 496.719,Z 443.31,A -85,B 0,C 180,E1 23872.791,E2 23872.791} C_VEL
LIN {X 0,Y 495.592,Z 459.692,A -85,B 0,C 180,E1 23871.728,E2 23871.728} C_VEL
LIN {X 0,Y 494.357,Z 475.248,A -85,B 0,C 180,E1 23870.48,E2 23870.48} C_VEL
LIN {X 0,Y 493.097,Z 489.847,A -85,B 0,C 180,E1 23869.053,E2 23869.053} C_VEL
LIN {X 0,Y 491.935,Z 502.988,A -85,B 0,C 180,E1 23867.505,E2 23867.505} C_VEL
LIN {X 0,Y 490.806,Z 515.546,A -85,B 0,C 180,E1 23865.72,E2 23865.72} C_VEL
LIN {X 0,Y 489.875,Z 526.56,A -85,B 0,C 180,E1 23863.815,E2 23863.815} C_VEL
LIN {X 0,Y 489.124,Z 536.431,A -85,B 0,C 180,E1 23861.716,E2 23861.716} C_VEL
LIN {X 0,Y 488.609,Z 544.567,A -85,B 0,C 180,E1 23859.54,E2 23859.54} C_VEL
LIN {X 0,Y 488.291,Z 551.013,A -85,B 0,C 180,E1 23857.293,E2 23857.293} C_VEL
LIN {X 0,Y 488.12,Z 555.625,A -85,B 0,C 180,E1 23855.052,E2 23855.052} C_VEL
LIN {X 0,Y 488.042,Z 558.631,A -85,B 0,C 180,E1 23852.7,E2 23852.7} C_VEL
LIN {X 0,Y 488.02,Z 559.805,A -85,B 0,C 180,E1 23850.469,E2 23850.469} C_VEL
LIN {X 0,Y 488.032,Z 559.37,A -85,B 0,C 180,E1 23848.238,E2 23848.238} C_VEL
LIN {X 0,Y 488.074,Z 557.317,A -85,B 0,C 180,E1 23846.005,E2 23846.005} C_VEL
LIN {X 0,Y 488.191,Z 553.588,A -85,B 0,C 180,E1 23843.768,E2 23843.768} C_VEL
LIN {X 0,Y 488.425,Z 548.096,A -85,B 0,C 180,E1 23841.523,E2 23841.523} C_VEL
LIN {X 0,Y 488.812,Z 541.132,A -85,B 0,C 180,E1 23839.391,E2 23839.391} C_VEL
LIN {X 0,Y 489.386,Z 532.79,A -85,B 0,C 180,E1 23837.372,E2 23837.372} C_VEL
LIN {X 0,Y 490.205,Z 522.47,A -85,B 0,C 180,E1 23835.349,E2 23835.349} C_VEL
LIN {X 0,Y 491.164,Z 511.361,A -85,B 0,C 180,E1 23833.562,E2 23833.562} C_VEL
LIN {X 0,Y 492.287,Z 498.873,A -85,B 0,C 180,E1 23831.895,E2 23831.895} C_VEL
LIN {X 0,Y 493.524,Z 484.905,A -85,B 0,C 180,E1 23830.347,E2 23830.347} C_VEL
LIN {X 0,Y 494.784,Z 469.943,A -85,B 0,C 180,E1 23828.98,E2 23828.98} C_VEL
LIN {X 0,Y 495.985,Z 454.038,A -85,B 0,C 180,E1 23827.791,E2 23827.791} C_VEL
LIN {X 0,Y 497.087,Z 437.174,A -85,B 0,C 180,E1 23826.781,E2 23826.781} C_VEL
LIN {X 0,Y 497.997,Z 419.902,A -85,B 0,C 180,E1 23825.978,E2 23825.978} C_VEL
LIN {X 0,Y 498.693,Z 401.148,A -85,B 0,C 180,E1 23825.34,E2 23825.34} C_VEL
LIN {X 0,Y 499.104,Z 382.106,A -85,B 0,C 180,E1 23824.922,E2 23824.922} C_VEL
LIN {X 0,Y 500.526,Z 192.531,A -85,B 0,C 180,E1 23822.207,E2 23822.207} C_VEL
LIN {X 0,Y 497.084,Z 173.858,A -85,B 0,C 180,E1 23821.659,E2 23821.659} C_VEL
LIN {X 0,Y 499.104,Z 137.648,A -85,B 0,C 180,E1 23818.365,E2 23818.365} C_VEL
LIN {X 0,Y 492.33,Z 118.334,A -85,B 0,C 180,E1 23815.908,E2 23815.908} C_VEL
LIN {X 0,Y 488.782,Z 108.6,A -85,B 0,C 180,E1 23814.59,E2 23814.59} C_VEL
LIN {X 0,Y 488.818,Z 108.567,A -85,B 0,C 180,E1 23811.1,E2 23811.1} C_VEL
LIN {X 0,Y 488.833,Z 108.593,A -85,B 0,C 180,E1 23807.547,E2 23807.547} C_VEL
LIN {X 0,Y 488.829,Z 108.589,A -85,B 0,C 180,E1 23803.9,E2 23803.9} C_VEL
LIN {X 0,Y 488.829,Z 108.596,A -85,B 0,C 180,E1 23800.267,E2 23800.267} C_VEL
LIN {X 0,Y 488.827,Z 108.597,A -85,B 0,C 180,E1 23796.675,E2 23796.675} C_VEL
LIN {X 0,Y 488.839,Z 108.799,A -85,B 0,C 180,E1 23794.01,E2 23794.01} C_VEL
LIN {X 0,Y 497.061,Z 133.274,A -85,B 0,C 180,E1 23791.361,E2 23791.361} C_VEL
LIN {X 0,Y 497.085,Z 141.514,A -85,B 0,C 180,E1 23790.658,E2 23790.658} C_VEL
LIN {X 0,Y 496.089,Z 180.449,A -85,B 0,C 180,E1 23787.459,E2 23787.459} C_VEL
LIN {X 0,Y 498.01,Z 193.617,A -85,B 0,C 180,E1 23787.117,E2 23787.117} C_VEL
LIN {X 0,Y 495.19,Z 390.108,A -85,B 0,C 180,E1 23783.908,E2 23783.908} C_VEL
LIN {X 0,Y 494.752,Z 409.492,A -85,B 0,C 180,E1 23783.371,E2 23783.371} C_VEL
LIN {X 0,Y 494.158,Z 427.62,A -85,B 0,C 180,E1 23782.651,E2 23782.651} C_VEL
LIN {X 0,Y 493.453,Z 444.681,A -85,B 0,C 180,E1 23781.765,E2 23781.765} C_VEL
LIN {X 0,Y 492.661,Z 461.396,A -85,B 0,C 180,E1 23780.673,E2 23780.673} C_VEL
LIN {X 0,Y 491.818,Z 477.397,A -85,B 0,C 180,E1 23779.385,E2 23779.385} C_VEL
LIN {X 0,Y 490.976,Z 492.443,A -85,B 0,C 180,E1 23777.909,E2 23777.909} C_VEL
LIN {X 0,Y 490.23,Z 505.673,A -85,B 0,C 180,E1 23776.348,E2 23776.348} C_VEL
LIN {X 0,Y 489.535,Z 518.299,A -85,B 0,C 180,E1 23774.55,E2 23774.55} C_VEL
LIN {X 0,Y 488.983,Z 529.325,A -85,B 0,C 180,E1 23772.638,E2 23772.638} C_VEL
LIN {X 0,Y 488.59,Z 538.261,A -85,B 0,C 180,E1 23770.733,E2 23770.733} C_VEL
LIN {X 0,Y 488.32,Z 545.816,A -85,B 0,C 180,E1 23768.715,E2 23768.715} C_VEL
LIN {X 0,Y 488.165,Z 551.609,A -85,B 0,C 180,E1 23766.705,E2 23766.705} C_VEL
LIN {X 0,Y 488.069,Z 556.014,A -85,B 0,C 180,E1 23764.583,E2 23764.583} C_VEL
LIN {X 0,Y 488.039,Z 558.748,A -85,B 0,C 180,E1 23762.466,E2 23762.466} C_VEL
LIN {X 0,Y 488.031,Z 559.892,A -85,B 0,C 180,E1 23760.352,E2 23760.352} C_VEL
LIN {X 0,Y 488.035,Z 559.467,A -85,B 0,C 180,E1 23758.239,E2 23758.239} C_VEL
LIN {X 0,Y 488.073,Z 557.412,A -85,B 0,C 180,E1 23756.085,E2 23756.085} C_VEL
LIN {X 0,Y 488.147,Z 553.823,A -85,B 0,C 180,E1 23754.004,E2 23754.004} C_VEL
LIN {X 0,Y 488.3,Z 548.434,A -85,B 0,C 180,E1 23751.878,E2 23751.878} C_VEL
LIN {X 0,Y 488.547,Z 541.579,A -85,B 0,C 180,E1 23749.863,E2 23749.863} C_VEL
LIN {X 0,Y 488.926,Z 532.801,A -85,B 0,C 180,E1 23747.841,E2 23747.841} C_VEL
LIN {X 0,Y 489.439,Z 522.459,A -85,B 0,C 180,E1 23745.931,E2 23745.931} C_VEL
LIN {X 0,Y 490.068,Z 510.514,A -85,B 0,C 180,E1 23744.134,E2 23744.134} C_VEL
LIN {X 0,Y 490.766,Z 497.387,A -85,B 0,C 180,E1 23742.512,E2 23742.512} C_VEL
LIN {X 0,Y 491.532,Z 482.625,A -85,B 0,C 180,E1 23741.006,E2 23741.006} C_VEL
LIN {X 0,Y 492.265,Z 467.537,A -85,B 0,C 180,E1 23739.739,E2 23739.739} C_VEL
LIN {X 0,Y 492.989,Z 450.539,A -85,B 0,C 180,E1 23738.58,E2 23738.58} C_VEL
LIN {X 0,Y 493.62,Z 432.617,A -85,B 0,C 180,E1 23737.617,E2 23737.617} C_VEL
LIN {X 0,Y 494.133,Z 414.329,A -85,B 0,C 180,E1 23736.867,E2 23736.867} C_VEL
LIN {X 0,Y 494.494,Z 395.246,A -85,B 0,C 180,E1 23736.313,E2 23736.313} C_VEL
LIN {X 0,Y 494.819,Z 365.111,A -85,B 0,C 180,E1 23735.791,E2 23735.791} C_VEL
LIN {X 0,Y 496.504,Z 258.993,A -85,B 0,C 180,E1 23733.998,E2 23733.998} C_VEL
LIN {X 0,Y 497.917,Z 191.175,A -85,B 0,C 180,E1 23732.741,E2 23732.741} C_VEL
LIN {X 0,Y 497.106,Z 186.005,A -85,B 0,C 180,E1 23732.574,E2 23732.574} C_VEL
LIN {X 0,Y 497.592,Z 147.436,A -85,B 0,C 180,E1 23729.578,E2 23729.578} C_VEL
LIN {X 0,Y 497.555,Z 132.574,A -85,B 0,C 180,E1 23728.436,E2 23728.436} C_VEL
LIN {X 0,Y 492.972,Z 118.735,A -85,B 0,C 180,E1 23727.001,E2 23727.001} C_VEL
LIN {X 0,Y 488.868,Z 108.969,A -85,B 0,C 180,E1 23725.884,E2 23725.884} C_VEL
LIN {X 0,Y 488.823,Z 108.598,A -85,B 0,C 180,E1 23725.772,E2 23725.772} C_VEL
LIN {X 0,Y 488.787,Z 108.6,A -85,B 0,C 180,E1 23722.293,E2 23722.293} C_VEL
LIN {X 0,Y 488.776,Z 108.601,A -85,B 0,C 180,E1 23718.8,E2 23718.8} C_VEL
LIN {X 0,Y 488.8,Z 108.601,A -85,B 0,C 180,E1 23715.386,E2 23715.386} C_VEL
LIN {X 0,Y 488.811,Z 108.598,A -85,B 0,C 180,E1 23711.824,E2 23711.824} C_VEL
LIN {X 0,Y 488.8,Z 108.816,A -85,B 0,C 180,E1 23709.257,E2 23709.257} C_VEL
LIN {X 0,Y 498.372,Z 132.613,A -85,B 0,C 180,E1 23706.544,E2 23706.544} C_VEL
LIN {X 0,Y 501.507,Z 140.661,A -85,B 0,C 180,E1 23705.681,E2 23705.681} C_VEL
LIN {X 0,Y 500.401,Z 164.23,A -85,B 0,C 180,E1 23703.989,E2 23703.989} C_VEL
LIN {X 0,Y 502.953,Z 182.908,A -85,B 0,C 180,E1 23703.499,E2 23703.499} C_VEL
LIN {X 0,Y 499.929,Z 400.766,A -85,B 0,C 180,E1 23700.089,E2 23700.089} C_VEL
LIN {X 0,Y 499.369,Z 429.482,A -85,B 0,C 180,E1 23699.579,E2 23699.579} C_VEL
LIN {X 0,Y 498.587,Z 450.908,A -85,B 0,C 180,E1 23698.98,E2 23698.98} C_VEL
LIN {X 0,Y 497.659,Z 470.965,A -85,B 0,C 180,E1 23698.207,E2 23698.207} C_VEL
LIN {X 0,Y 496.633,Z 489.993,A -85,B 0,C 180,E1 23697.267,E2 23697.267} C_VEL
LIN {X 0,Y 495.376,Z 509.785,A -85,B 0,C 180,E1 23696.047,E2 23696.047} C_VEL
LIN {X 0,Y 494.135,Z 528.514,A -85,B 0,C 180,E1 23694.635,E2 23694.635} C_VEL
LIN {X 0,Y 492.939,Z 545.433,A -85,B 0,C 180,E1 23693.11,E2 23693.11} C_VEL
LIN {X 0,Y 491.841,Z 560.93,A -85,B 0,C 180,E1 23691.465,E2 23691.465} C_VEL
LIN {X 0,Y 490.82,Z 575.571,A -85,B 0,C 180,E1 23689.642,E2 23689.642} C_VEL
LIN {X 0,Y 490.1,Z 586.34,A -85,B 0,C 180,E1 23688.066,E2 23688.066} C_VEL
LIN {X 0,Y 489.324,Z 598.004,A -85,B 0,C 180,E1 23686.013,E2 23686.013} C_VEL
LIN {X 0,Y 488.709,Z 608.842,A -85,B 0,C 180,E1 23683.73,E2 23683.73} C_VEL
LIN {X 0,Y 488.319,Z 617.652,A -85,B 0,C 180,E1 23681.457,E2 23681.457} C_VEL
LIN {X 0,Y 488.092,Z 624.682,A -85,B 0,C 180,E1 23679.195,E2 23679.195} C_VEL
LIN {X 0,Y 487.97,Z 630.258,A -85,B 0,C 180,E1 23676.826,E2 23676.826} C_VEL
LIN {X 0,Y 487.912,Z 634.085,A -85,B 0,C 180,E1 23674.467,E2 23674.467} C_VEL
LIN {X 0,Y 487.907,Z 636.303,A -85,B 0,C 180,E1 23672.115,E2 23672.115} C_VEL
LIN {X 0,Y 487.906,Z 636.962,A -85,B 0,C 180,E1 23669.766,E2 23669.766} C_VEL
LIN {X 0,Y 487.905,Z 636.031,A -85,B 0,C 180,E1 23667.417,E2 23667.417} C_VEL
LIN {X 0,Y 487.928,Z 633.447,A -85,B 0,C 180,E1 23665.063,E2 23665.063} C_VEL
LIN {X 0,Y 487.982,Z 629.245,A -85,B 0,C 180,E1 23662.702,E2 23662.702} C_VEL
LIN {X 0,Y 488.124,Z 623.328,A -85,B 0,C 180,E1 23660.331,E2 23660.331} C_VEL
LIN {X 0,Y 488.382,Z 616.011,A -85,B 0,C 180,E1 23658.067,E2 23658.067} C_VEL
LIN {X 0,Y 488.816,Z 606.791,A -85,B 0,C 180,E1 23655.792,E2 23655.792} C_VEL
LIN {X 0,Y 489.442,Z 596.108,A -85,B 0,C 180,E1 23653.626,E2 23653.626} C_VEL
LIN {X 0,Y 490.256,Z 584.021,A -85,B 0,C 180,E1 23651.573,E2 23651.573} C_VEL
LIN {X 0,Y 491.141,Z 570.985,A -85,B 0,C 180,E1 23649.753,E2 23649.753} C_VEL
LIN {X 0,Y 492.209,Z 555.938,A -85,B 0,C 180,E1 23647.97,E2 23647.97} C_VEL
LIN {X 0,Y 493.396,Z 539.09,A -85,B 0,C 180,E1 23646.282,E2 23646.282} C_VEL
LIN {X 0,Y 494.654,Z 520.861,A -85,B 0,C 180,E1 23644.755,E2 23644.755} C_VEL
LIN {X 0,Y 495.854,Z 502.397,A -85,B 0,C 180,E1 23643.473,E2 23643.473} C_VEL
LIN {X 0,Y 496.973,Z 483.624,A -85,B 0,C 180,E1 23642.4,E2 23642.4} C_VEL
LIN {X 0,Y 498.01,Z 463.714,A -85,B 0,C 180,E1 23641.49,E2 23641.49} C_VEL
LIN {X 0,Y 498.901,Z 443.142,A -85,B 0,C 180,E1 23640.776,E2 23640.776} C_VEL
LIN {X 0,Y 499.566,Z 422.588,A -85,B 0,C 180,E1 23640.271,E2 23640.271} C_VEL
LIN {X 0,Y 502.815,Z 191.299,A -85,B 0,C 180,E1 23636.634,E2 23636.634} C_VEL
LIN {X 0,Y 502.767,Z 180.177,A -85,B 0,C 180,E1 23636.443,E2 23636.443} C_VEL
LIN {X 0,Y 500.331,Z 163.36,A -85,B 0,C 180,E1 23635.976,E2 23635.976} C_VEL
LIN {X 0,Y 501.514,Z 140.688,A -85,B 0,C 180,E1 23634.322,E2 23634.322} C_VEL
LIN {X 0,Y 492.661,Z 118.263,A -85,B 0,C 180,E1 23631.853,E2 23631.853} C_VEL
LIN {X 0,Y 488.797,Z 108.704,A -85,B 0,C 180,E1 23630.736,E2 23630.736} C_VEL
LIN {X 0,Y 488.776,Z 108.601,A -85,B 0,C 180,E1 23627.224,E2 23627.224} C_VEL
LIN {X 0,Y 488.802,Z 108.592,A -85,B 0,C 180,E1 23623.74,E2 23623.74} C_VEL
LIN {X 0,Y 488.827,Z 108.579,A -85,B 0,C 180,E1 23620.267,E2 23620.267} C_VEL
LIN {X 0,Y 488.781,Z 108.584,A -85,B 0,C 180,E1 23616.824,E2 23616.824} C_VEL
LIN {X 0,Y 488.772,Z 108.59,A -85,B 0,C 180,E1 23613.246,E2 23613.246} C_VEL
LIN {X 0,Y 488.796,Z 108.593,A -85,B 0,C 180,E1 23609.806,E2 23609.806} C_VEL
LIN {X 0,Y 488.822,Z 108.597,A -85,B 0,C 180,E1 23606.35,E2 23606.35} C_VEL
LIN {X 0,Y 488.78,Z 108.591,A -85,B 0,C 180,E1 23602.871,E2 23602.871} C_VEL
LIN {X 0,Y 488.768,Z 108.588,A -85,B 0,C 180,E1 23599.353,E2 23599.353} C_VEL
LIN {X 0,Y 488.792,Z 108.599,A -85,B 0,C 180,E1 23595.909,E2 23595.909} C_VEL
LIN {X 0,Y 488.812,Z 108.582,A -85,B 0,C 180,E1 23592.522,E2 23592.522} C_VEL
LIN {X 0,Y 488.772,Z 108.597,A -85,B 0,C 180,E1 23589.062,E2 23589.062} C_VEL
LIN {X 0,Y 488.765,Z 108.596,A -85,B 0,C 180,E1 23585.517,E2 23585.517} C_VEL
LIN {X 0,Y 488.796,Z 108.587,A -85,B 0,C 180,E1 23582.11,E2 23582.11} C_VEL
LIN {X 0,Y 488.802,Z 108.594,A -85,B 0,C 180,E1 23578.71,E2 23578.71} C_VEL
LIN {X 0,Y 488.761,Z 108.59,A -85,B 0,C 180,E1 23575.306,E2 23575.306} C_VEL
LIN {X 0,Y 488.763,Z 108.6,A -85,B 0,C 180,E1 23571.648,E2 23571.648} C_VEL
LIN {X 0,Y 488.793,Z 108.586,A -85,B 0,C 180,E1 23568.196,E2 23568.196} C_VEL
LIN {X 0,Y 488.811,Z 108.599,A -85,B 0,C 180,E1 23564.7,E2 23564.7} C_VEL
LIN {X 0,Y 488.765,Z 108.591,A -85,B 0,C 180,E1 23561.266,E2 23561.266} C_VEL
LIN {X 0,Y 488.76,Z 108.592,A -85,B 0,C 180,E1 23557.762,E2 23557.762} C_VEL
LIN {X 0,Y 488.792,Z 108.599,A -85,B 0,C 180,E1 23554.3,E2 23554.3} C_VEL
LIN {X 0,Y 488.802,Z 108.585,A -85,B 0,C 180,E1 23550.859,E2 23550.859} C_VEL
LIN {X 0,Y 488.759,Z 108.594,A -85,B 0,C 180,E1 23547.439,E2 23547.439} C_VEL
LIN {X 0,Y 488.757,Z 108.598,A -85,B 0,C 180,E1 23543.902,E2 23543.902} C_VEL
LIN {X 0,Y 488.794,Z 108.599,A -85,B 0,C 180,E1 23540.458,E2 23540.458} C_VEL
LIN {X 0,Y 488.785,Z 108.601,A -85,B 0,C 180,E1 23537.063,E2 23537.063} C_VEL
LIN {X 0,Y 488.754,Z 108.602,A -85,B 0,C 180,E1 23533.582,E2 23533.582} C_VEL
LIN {X 0,Y 488.755,Z 108.599,A -85,B 0,C 180,E1 23529.967,E2 23529.967} C_VEL
LIN {X 0,Y 488.807,Z 108.602,A -85,B 0,C 180,E1 23526.675,E2 23526.675} C_VEL
LIN {X 0,Y 488.78,Z 108.644,A -85,B 0,C 180,E1 23525.293,E2 23525.293} C_VEL
LIN {X 0,Y 495.655,Z 127.638,A -85,B 0,C 180,E1 23522.793,E2 23522.793} C_VEL
LIN {X 0,Y 496.247,Z 132.457,A -85,B 0,C 180,E1 23522.27,E2 23522.27} C_VEL
LIN {X 0,Y 495.033,Z 139.614,A -85,B 0,C 180,E1 23521.664,E2 23521.664} C_VEL
LIN {X 0,Y 491.239,Z 153.629,A -85,B 0,C 180,E1 23520.586,E2 23520.586} C_VEL
LIN {X 0,Y 490.924,Z 156.369,A -85,B 0,C 180,E1 23520.345,E2 23520.345} C_VEL
LIN {X 0,Y 489.994,Z 174.481,A -85,B 0,C 180,E1 23518.718,E2 23518.718} C_VEL
LIN {X 0,Y 493.735,Z 195.654,A -85,B 0,C 180,E1 23518.118,E2 23518.118} C_VEL
LIN {X 0,Y 491.972,Z 388.764,A -85,B 0,C 180,E1 23515.312,E2 23515.312} C_VEL
LIN {X 0,Y 491.42,Z 407.795,A -85,B 0,C 180,E1 23514.814,E2 23514.814} C_VEL
LIN {X 0,Y 490.595,Z 425.952,A -85,B 0,C 180,E1 23514.118,E2 23514.118} C_VEL
LIN {X 0,Y 489.532,Z 443.512,A -85,B 0,C 180,E1 23513.215,E2 23513.215} C_VEL
LIN {X 0,Y 488.314,Z 460.058,A -85,B 0,C 180,E1 23512.132,E2 23512.132} C_VEL
LIN {X 0,Y 486.992,Z 475.67,A -85,B 0,C 180,E1 23510.867,E2 23510.867} C_VEL
LIN {X 0,Y 485.675,Z 489.979,A -85,B 0,C 180,E1 23509.458,E2 23509.458} C_VEL
LIN {X 0,Y 484.34,Z 503.951,A -85,B 0,C 180,E1 23507.789,E2 23507.789} C_VEL
LIN {X 0,Y 483.127,Z 516.475,A -85,B 0,C 180,E1 23505.976,E2 23505.976} C_VEL
LIN {X 0,Y 482.12,Z 527.47,A -85,B 0,C 180,E1 23504.042,E2 23504.042} C_VEL
LIN {X 0,Y 481.324,Z 536.982,A -85,B 0,C 180,E1 23501.989,E2 23501.989} C_VEL
LIN {X 0,Y 480.749,Z 544.998,A -85,B 0,C 180,E1 23499.819,E2 23499.819} C_VEL
LIN {X 0,Y 480.395,Z 551.19,A -85,B 0,C 180,E1 23497.654,E2 23497.654} C_VEL
LIN {X 0,Y 480.183,Z 555.935,A -85,B 0,C 180,E1 23495.376,E2 23495.376} C_VEL
LIN {X 0,Y 480.082,Z 558.974,A -85,B 0,C 180,E1 23493.103,E2 23493.103} C_VEL
LIN {X 0,Y 480.053,Z 560.388,A -85,B 0,C 180,E1 23490.835,E2 23490.835} C_VEL
LIN {X 0,Y 480.055,Z 560.213,A -85,B 0,C 180,E1 23488.567,E2 23488.567} C_VEL
LIN {X 0,Y 480.098,Z 558.442,A -85,B 0,C 180,E1 23486.298,E2 23486.298} C_VEL
LIN {X 0,Y 480.222,Z 555.024,A -85,B 0,C 180,E1 23484.024,E2 23484.024} C_VEL
LIN {X 0,Y 480.464,Z 549.872,A -85,B 0,C 180,E1 23481.744,E2 23481.744} C_VEL
LIN {X 0,Y 480.861,Z 543.272,A -85,B 0,C 180,E1 23479.577,E2 23479.577} C_VEL
LIN {X 0,Y 481.457,Z 535.308,A -85,B 0,C 180,E1 23477.526,E2 23477.526} C_VEL
LIN {X 0,Y 482.304,Z 525.378,A -85,B 0,C 180,E1 23475.472,E2 23475.472} C_VEL
LIN {X 0,Y 483.295,Z 514.713,A -85,B 0,C 180,E1 23473.658,E2 23473.658} C_VEL
LIN {X 0,Y 484.456,Z 502.758,A -85,B 0,C 180,E1 23471.965,E2 23471.965} C_VEL
LIN {X 0,Y 485.76,Z 489.067,A -85,B 0,C 180,E1 23470.355,E2 23470.355} C_VEL
LIN {X 0,Y 487.089,Z 474.604,A -85,B 0,C 180,E1 23468.947,E2 23468.947} C_VEL
LIN {X 0,Y 488.414,Z 458.843,A -85,B 0,C 180,E1 23467.688,E2 23467.688} C_VEL
LIN {X 0,Y 489.649,Z 441.873,A -85,B 0,C 180,E1 23466.598,E2 23466.598} C_VEL
LIN {X 0,Y 490.685,Z 424.483,A -85,B 0,C 180,E1 23465.725,E2 23465.725} C_VEL
LIN {X 0,Y 491.489,Z 405.9,A -85,B 0,C 180,E1 23465.034,E2 23465.034} C_VEL
LIN {X 0,Y 492.008,Z 386.991,A -85,B 0,C 180,E1 23464.564,E2 23464.564} C_VEL
LIN {X 0,Y 493.63,Z 193.801,A -85,B 0,C 180,E1 23461.751,E2 23461.751} C_VEL
LIN {X 0,Y 489.964,Z 173.656,A -85,B 0,C 180,E1 23461.143,E2 23461.143} C_VEL
LIN {X 0,Y 491.953,Z 140.622,A -85,B 0,C 180,E1 23458.1,E2 23458.1} C_VEL
LIN {X 0,Y 485.239,Z 121.554,A -85,B 0,C 180,E1 23455.625,E2 23455.625} C_VEL
LIN {X 0,Y 480.85,Z 109.59,A -85,B 0,C 180,E1 23453.952,E2 23453.952} C_VEL
LIN {X 0,Y 480.849,Z 109.559,A -85,B 0,C 180,E1 23450.484,E2 23450.484} C_VEL
LIN {X 0,Y 480.875,Z 109.58,A -85,B 0,C 180,E1 23447,E2 23447} C_VEL
LIN {X 0,Y 480.891,Z 109.575,A -85,B 0,C 180,E1 23443.478,E2 23443.478} C_VEL
LIN {X 0,Y 480.884,Z 109.585,A -85,B 0,C 180,E1 23439.822,E2 23439.822} C_VEL
LIN {X 0,Y 480.883,Z 109.585,A -85,B 0,C 180,E1 23436.193,E2 23436.193} C_VEL
LIN {X 0,Y 480.9,Z 109.694,A -85,B 0,C 180,E1 23434.496,E2 23434.496} C_VEL
LIN {X 0,Y 489.713,Z 135.803,A -85,B 0,C 180,E1 23431.635,E2 23431.635} C_VEL
LIN {X 0,Y 489.958,Z 138.843,A -85,B 0,C 180,E1 23431.358,E2 23431.358} C_VEL
LIN {X 0,Y 488.734,Z 178.156,A -85,B 0,C 180,E1 23428.069,E2 23428.069} C_VEL
LIN {X 0,Y 488.773,Z 180.916,A -85,B 0,C 180,E1 23427.873,E2 23427.873} C_VEL
LIN {X 0,Y 490.791,Z 194.743,A -85,B 0,C 180,E1 23427.505,E2 23427.505} C_VEL
LIN {X 0,Y 487.715,Z 390.652,A -85,B 0,C 180,E1 23424.234,E2 23424.234} C_VEL
LIN {X 0,Y 487.244,Z 410.141,A -85,B 0,C 180,E1 23423.684,E2 23423.684} C_VEL
LIN {X 0,Y 486.578,Z 428.977,A -85,B 0,C 180,E1 23422.917,E2 23422.917} C_VEL
LIN {X 0,Y 485.817,Z 446.192,A -85,B 0,C 180,E1 23421.998,E2 23421.998} C_VEL
LIN {X 0,Y 484.982,Z 462.654,A -85,B 0,C 180,E1 23420.896,E2 23420.896} C_VEL
LIN {X 0,Y 484.135,Z 477.873,A -85,B 0,C 180,E1 23419.651,E2 23419.651} C_VEL
LIN {X 0,Y 483.271,Z 492.5,A -85,B 0,C 180,E1 23418.205,E2 23418.205} C_VEL
LIN {X 0,Y 482.465,Z 505.859,A -85,B 0,C 180,E1 23416.618,E2 23416.618} C_VEL
LIN {X 0,Y 481.759,Z 517.828,A -85,B 0,C 180,E1 23414.913,E2 23414.913} C_VEL
LIN {X 0,Y 481.183,Z 528.44,A -85,B 0,C 180,E1 23413.091,E2 23413.091} C_VEL
LIN {X 0,Y 480.707,Z 538.199,A -85,B 0,C 180,E1 23411.032,E2 23411.032} C_VEL
LIN {X 0,Y 480.399,Z 545.923,A -85,B 0,C 180,E1 23408.981,E2 23408.981} C_VEL
LIN {X 0,Y 480.209,Z 552.17,A -85,B 0,C 180,E1 23406.816,E2 23406.816} C_VEL
LIN {X 0,Y 480.103,Z 556.618,A -85,B 0,C 180,E1 23404.659,E2 23404.659} C_VEL
LIN {X 0,Y 480.067,Z 559.386,A -85,B 0,C 180,E1 23402.507,E2 23402.507} C_VEL
LIN {X 0,Y 480.058,Z 560.552,A -85,B 0,C 180,E1 23400.358,E2 23400.358} C_VEL
LIN {X 0,Y 480.064,Z 560.138,A -85,B 0,C 180,E1 23398.21,E2 23398.21} C_VEL
LIN {X 0,Y 480.111,Z 558.042,A -85,B 0,C 180,E1 23395.991,E2 23395.991} C_VEL
LIN {X 0,Y 480.205,Z 554.227,A -85,B 0,C 180,E1 23393.785,E2 23393.785} C_VEL
LIN {X 0,Y 480.376,Z 548.718,A -85,B 0,C 180,E1 23391.623,E2 23391.623} C_VEL
LIN {X 0,Y 480.667,Z 541.721,A -85,B 0,C 180,E1 23389.574,E2 23389.574} C_VEL
LIN {X 0,Y 481.095,Z 532.761,A -85,B 0,C 180,E1 23387.518,E2 23387.518} C_VEL
LIN {X 0,Y 481.657,Z 522.156,A -85,B 0,C 180,E1 23385.576,E2 23385.576} C_VEL
LIN {X 0,Y 482.347,Z 509.932,A -85,B 0,C 180,E1 23383.749,E2 23383.749} C_VEL
LIN {X 0,Y 483.117,Z 496.539,A -85,B 0,C 180,E1 23382.102,E2 23382.102} C_VEL
LIN {X 0,Y 483.953,Z 481.403,A -85,B 0,C 180,E1 23380.572,E2 23380.572} C_VEL
LIN {X 0,Y 484.74,Z 465.985,A -85,B 0,C 180,E1 23379.296,E2 23379.296} C_VEL
LIN {X 0,Y 485.494,Z 449.41,A -85,B 0,C 180,E1 23378.178,E2 23378.178} C_VEL
LIN {X 0,Y 486.136,Z 432.12,A -85,B 0,C 180,E1 23377.253,E2 23377.253} C_VEL
LIN {X 0,Y 486.677,Z 413.355,A -85,B 0,C 180,E1 23376.492,E2 23376.492} C_VEL
LIN {X 0,Y 487.033,Z 393.931,A -85,B 0,C 180,E1 23375.948,E2 23375.948} C_VEL
LIN {X 0,Y 489.17,Z 265.973,A -85,B 0,C 180,E1 23373.711,E2 23373.711} C_VEL
LIN {X 0,Y 490.965,Z 192.44,A -85,B 0,C 180,E1 23372.299,E2 23372.299} C_VEL
LIN {X 0,Y 490.147,Z 186.761,A -85,B 0,C 180,E1 23372.085,E2 23372.085} C_VEL
LIN {X 0,Y 490.725,Z 148.223,A -85,B 0,C 180,E1 23369.071,E2 23369.071} C_VEL
LIN {X 0,Y 490.676,Z 135.463,A -85,B 0,C 180,E1 23368.072,E2 23368.072} C_VEL
LIN {X 0,Y 486.128,Z 122.023,A -85,B 0,C 180,E1 23366.622,E2 23366.622} C_VEL
LIN {X 0,Y 482.158,Z 113.009,A -85,B 0,C 180,E1 23365.52,E2 23365.52} C_VEL
LIN {X 0,Y 480.872,Z 109.589,A -85,B 0,C 180,E1 23365.088,E2 23365.088} C_VEL
LIN {X 0,Y 480.894,Z 109.586,A -85,B 0,C 180,E1 23361.562,E2 23361.562} C_VEL
LIN {X 0,Y 480.865,Z 109.589,A -85,B 0,C 180,E1 23357.969,E2 23357.969} C_VEL
LIN {X 0,Y 480.828,Z 109.592,A -85,B 0,C 180,E1 23354.49,E2 23354.49} C_VEL
LIN {X 0,Y 480.821,Z 109.593,A -85,B 0,C 180,E1 23350.923,E2 23350.923} C_VEL
LIN {X 0,Y 480.896,Z 109.756,A -85,B 0,C 180,E1 23349.896,E2 23349.896} C_VEL
LIN {X 0,Y 490.842,Z 134.303,A -85,B 0,C 180,E1 23347.012,E2 23347.012} C_VEL
LIN {X 0,Y 494.428,Z 144.154,A -85,B 0,C 180,E1 23345.95,E2 23345.95} C_VEL
LIN {X 0,Y 493.387,Z 164.415,A -85,B 0,C 180,E1 23344.478,E2 23344.478} C_VEL
LIN {X 0,Y 496.036,Z 184.116,A -85,B 0,C 180,E1 23343.947,E2 23343.947} C_VEL
LIN {X 0,Y 492.252,Z 424.041,A -85,B 0,C 180,E1 23340.085,E2 23340.085} C_VEL
LIN {X 0,Y 491.451,Z 445.684,A -85,B 0,C 180,E1 23339.522,E2 23339.522} C_VEL
LIN {X 0,Y 490.431,Z 467.087,A -85,B 0,C 180,E1 23338.727,E2 23338.727} C_VEL
LIN {X 0,Y 489.281,Z 486.845,A -85,B 0,C 180,E1 23337.768,E2 23337.768} C_VEL
LIN {X 0,Y 488.029,Z 506.122,A -85,B 0,C 180,E1 23336.602,E2 23336.602} C_VEL
LIN {X 0,Y 486.789,Z 523.949,A -85,B 0,C 180,E1 23335.293,E2 23335.293} C_VEL
LIN {X 0,Y 485.466,Z 541.559,A -85,B 0,C 180,E1 23333.745,E2 23333.745} C_VEL
LIN {X 0,Y 484.272,Z 557.618,A -85,B 0,C 180,E1 23332.073,E2 23332.073} C_VEL
LIN {X 0,Y 483.152,Z 572.725,A -85,B 0,C 180,E1 23330.219,E2 23330.219} C_VEL
LIN {X 0,Y 482.141,Z 587.072,A -85,B 0,C 180,E1 23328.124,E2 23328.124} C_VEL
LIN {X 0,Y 481.33,Z 599.691,A -85,B 0,C 180,E1 23325.915,E2 23325.915} C_VEL
LIN {X 0,Y 480.796,Z 608.841,A -85,B 0,C 180,E1 23323.96,E2 23323.96} C_VEL
LIN {X 0,Y 480.365,Z 617.651,A -85,B 0,C 180,E1 23321.649,E2 23321.649} C_VEL
LIN {X 0,Y 480.113,Z 624.682,A -85,B 0,C 180,E1 23319.349,E2 23319.349} C_VEL
LIN {X 0,Y 479.979,Z 630.258,A -85,B 0,C 180,E1 23316.94,E2 23316.94} C_VEL
LIN {X 0,Y 479.914,Z 634.085,A -85,B 0,C 180,E1 23314.542,E2 23314.542} C_VEL
LIN {X 0,Y 479.906,Z 636.303,A -85,B 0,C 180,E1 23312.15,E2 23312.15} C_VEL
LIN {X 0,Y 479.906,Z 636.962,A -85,B 0,C 180,E1 23309.762,E2 23309.762} C_VEL
LIN {X 0,Y 479.907,Z 636.03,A -85,B 0,C 180,E1 23307.374,E2 23307.374} C_VEL
LIN {X 0,Y 479.929,Z 633.446,A -85,B 0,C 180,E1 23304.981,E2 23304.981} C_VEL
LIN {X 0,Y 479.991,Z 629.165,A -85,B 0,C 180,E1 23302.542,E2 23302.542} C_VEL
LIN {X 0,Y 480.147,Z 623.328,A -85,B 0,C 180,E1 23300.169,E2 23300.169} C_VEL
LIN {X 0,Y 480.431,Z 616.011,A -85,B 0,C 180,E1 23297.867,E2 23297.867} C_VEL
LIN {X 0,Y 480.914,Z 606.788,A -85,B 0,C 180,E1 23295.554,E2 23295.554} C_VEL
LIN {X 0,Y 481.483,Z 597.049,A -85,B 0,C 180,E1 23293.596,E2 23293.596} C_VEL
LIN {X 0,Y 482.297,Z 584.674,A -85,B 0,C 180,E1 23291.508,E2 23291.508} C_VEL
LIN {X 0,Y 483.281,Z 570.828,A -85,B 0,C 180,E1 23289.535,E2 23289.535} C_VEL
LIN {X 0,Y 484.44,Z 555.451,A -85,B 0,C 180,E1 23287.682,E2 23287.682} C_VEL
LIN {X 0,Y 485.727,Z 538.389,A -85,B 0,C 180,E1 23285.948,E2 23285.948} C_VEL
LIN {X 0,Y 487.069,Z 520.13,A -85,B 0,C 180,E1 23284.399,E2 23284.399} C_VEL
LIN {X 0,Y 488.343,Z 501.54,A -85,B 0,C 180,E1 23283.098,E2 23283.098} C_VEL
LIN {X 0,Y 489.492,Z 483.361,A -85,B 0,C 180,E1 23282.05,E2 23282.05} C_VEL
LIN {X 0,Y 490.602,Z 463.279,A -85,B 0,C 180,E1 23281.119,E2 23281.119} C_VEL
LIN {X 0,Y 491.565,Z 442.895,A -85,B 0,C 180,E1 23280.398,E2 23280.398} C_VEL
LIN {X 0,Y 492.289,Z 422.301,A -85,B 0,C 180,E1 23279.88,E2 23279.88} C_VEL
LIN {X 0,Y 496.055,Z 183.247,A -85,B 0,C 180,E1 23276.038,E2 23276.038} C_VEL
LIN {X 0,Y 493.301,Z 163.592,A -85,B 0,C 180,E1 23275.494,E2 23275.494} C_VEL
LIN {X 0,Y 494.362,Z 143.569,A -85,B 0,C 180,E1 23273.999,E2 23273.999} C_VEL
LIN {X 0,Y 486.005,Z 122.285,A -85,B 0,C 180,E1 23271.612,E2 23271.612} C_VEL
LIN {X 0,Y 481.098,Z 110.647,A -85,B 0,C 180,E1 23270.201,E2 23270.201} C_VEL
LIN {X 0,Y 480.898,Z 109.58,A -85,B 0,C 180,E1 23270.061,E2 23270.061} C_VEL
LIN {X 0,Y 480.862,Z 109.585,A -85,B 0,C 180,E1 23266.51,E2 23266.51} C_VEL
LIN {X 0,Y 480.837,Z 109.581,A -85,B 0,C 180,E1 23263.004,E2 23263.004} C_VEL
LIN {X 0,Y 480.833,Z 109.556,A -85,B 0,C 180,E1 23259.328,E2 23259.328} C_VEL
LIN {X 0,Y 480.86,Z 109.583,A -85,B 0,C 180,E1 23255.815,E2 23255.815} C_VEL
LIN {X 0,Y 480.883,Z 109.575,A -85,B 0,C 180,E1 23252.3,E2 23252.3} C_VEL
LIN {X 0,Y 480.842,Z 109.579,A -85,B 0,C 180,E1 23248.843,E2 23248.843} C_VEL
LIN {X 0,Y 480.832,Z 109.585,A -85,B 0,C 180,E1 23245.364,E2 23245.364} C_VEL
LIN {X 0,Y 480.855,Z 109.589,A -85,B 0,C 180,E1 23241.851,E2 23241.851} C_VEL
LIN {X 0,Y 480.882,Z 109.572,A -85,B 0,C 180,E1 23238.298,E2 23238.298} C_VEL
LIN {X 0,Y 480.849,Z 109.586,A -85,B 0,C 180,E1 23234.786,E2 23234.786} C_VEL
LIN {X 0,Y 480.827,Z 109.586,A -85,B 0,C 180,E1 23231.272,E2 23231.272} C_VEL
LIN {X 0,Y 480.83,Z 109.573,A -85,B 0,C 180,E1 23227.648,E2 23227.648} C_VEL
LIN {X 0,Y 480.866,Z 109.589,A -85,B 0,C 180,E1 23224.173,E2 23224.173} C_VEL
LIN {X 0,Y 480.873,Z 109.569,A -85,B 0,C 180,E1 23220.595,E2 23220.595} C_VEL
LIN {X 0,Y 480.831,Z 109.588,A -85,B 0,C 180,E1 23217.139,E2 23217.139} C_VEL
LIN {X 0,Y 480.821,Z 109.581,A -85,B 0,C 180,E1 23213.552,E2 23213.552} C_VEL
LIN {X 0,Y 480.855,Z 109.582,A -85,B 0,C 180,E1 23210.183,E2 23210.183} C_VEL
LIN {X 0,Y 480.872,Z 109.579,A -85,B 0,C 180,E1 23206.656,E2 23206.656} C_VEL
LIN {X 0,Y 480.828,Z 109.582,A -85,B 0,C 180,E1 23203.199,E2 23203.199} C_VEL
LIN {X 0,Y 480.821,Z 109.589,A -85,B 0,C 180,E1 23199.679,E2 23199.679} C_VEL
LIN {X 0,Y 480.843,Z 109.578,A -85,B 0,C 180,E1 23196.193,E2 23196.193} C_VEL
LIN {X 0,Y 480.877,Z 109.576,A -85,B 0,C 180,E1 23192.6,E2 23192.6} C_VEL
LIN {X 0,Y 480.838,Z 109.588,A -85,B 0,C 180,E1 23189.095,E2 23189.095} C_VEL
LIN {X 0,Y 480.818,Z 109.587,A -85,B 0,C 180,E1 23185.554,E2 23185.554} C_VEL
LIN {X 0,Y 480.818,Z 109.588,A -85,B 0,C 180,E1 23181.858,E2 23181.858} C_VEL
LIN {X 0,Y 480.851,Z 109.584,A -85,B 0,C 180,E1 23178.447,E2 23178.447} C_VEL
LIN {X 0,Y 480.866,Z 109.583,A -85,B 0,C 180,E1 23174.843,E2 23174.843} C_VEL
LIN {X 0,Y 480.828,Z 109.592,A -85,B 0,C 180,E1 23171.35,E2 23171.35} C_VEL
LIN {X 0,Y 480.815,Z 109.587,A -85,B 0,C 180,E1 23167.838,E2 23167.838} C_VEL
LIN {X 0,Y 480.838,Z 109.745,A -85,B 0,C 180,E1 23165.9,E2 23165.9} C_VEL
LIN {X 0,Y 488.835,Z 131.575,A -85,B 0,C 180,E1 23162.956,E2 23162.956} C_VEL
LIN {X 0,Y 491.917,Z 141.063,A -85,B 0,C 180,E1 23161.764,E2 23161.764} C_VEL
LIN {X 0,Y 490.924,Z 156.369,A -85,B 0,C 180,E1 23160.345,E2 23160.345} C_VEL
LIN {X 0,Y 489.721,Z 161.119,A -85,B 0,C 180,E1 23159.985,E2 23159.985} C_VEL
LIN {X 0,Y 483.668,Z 173.008,A -85,B 0,C 180,E1 23159.312,E2 23159.312} C_VEL
LIN {X 0,Y 483.355,Z 176.82,A -85,B 0,C 180,E1 23159.166,E2 23159.166} C_VEL
LIN {X 0,Y 486.872,Z 196.991,A -85,B 0,C 180,E1 23158.584,E2 23158.584} C_VEL
LIN {X 0,Y 484.936,Z 389.224,A -85,B 0,C 180,E1 23155.754,E2 23155.754} C_VEL
LIN {X 0,Y 484.346,Z 408.232,A -85,B 0,C 180,E1 23155.252,E2 23155.252} C_VEL
LIN {X 0,Y 483.489,Z 426.104,A -85,B 0,C 180,E1 23154.56,E2 23154.56} C_VEL
LIN {X 0,Y 482.356,Z 443.749,A -85,B 0,C 180,E1 23153.646,E2 23153.646} C_VEL
LIN {X 0,Y 481.052,Z 460.361,A -85,B 0,C 180,E1 23152.548,E2 23152.548} C_VEL
LIN {X 0,Y 479.642,Z 476.028,A -85,B 0,C 180,E1 23151.266,E2 23151.266} C_VEL
LIN {X 0,Y 478.136,Z 491.257,A -85,B 0,C 180,E1 23149.737,E2 23149.737} C_VEL
LIN {X 0,Y 476.745,Z 504.84,A -85,B 0,C 180,E1 23148.082,E2 23148.082} C_VEL
LIN {X 0,Y 475.445,Z 517.325,A -85,B 0,C 180,E1 23146.241,E2 23146.241} C_VEL
LIN {X 0,Y 474.358,Z 528.286,A -85,B 0,C 180,E1 23144.276,E2 23144.276} C_VEL
LIN {X 0,Y 473.493,Z 537.769,A -85,B 0,C 180,E1 23142.19,E2 23142.19} C_VEL
LIN {X 0,Y 472.861,Z 545.757,A -85,B 0,C 180,E1 23139.984,E2 23139.984} C_VEL
LIN {X 0,Y 472.471,Z 551.918,A -85,B 0,C 180,E1 23137.783,E2 23137.783} C_VEL
LIN {X 0,Y 472.23,Z 556.625,A -85,B 0,C 180,E1 23135.467,E2 23135.467} C_VEL
LIN {X 0,Y 472.113,Z 559.634,A -85,B 0,C 180,E1 23133.156,E2 23133.156} C_VEL
LIN {X 0,Y 472.079,Z 561.034,A -85,B 0,C 180,E1 23130.849,E2 23130.849} C_VEL
LIN {X 0,Y 472.082,Z 560.863,A -85,B 0,C 180,E1 23128.543,E2 23128.543} C_VEL
LIN {X 0,Y 472.135,Z 559.114,A -85,B 0,C 180,E1 23126.235,E2 23126.235} C_VEL
LIN {X 0,Y 472.275,Z 555.731,A -85,B 0,C 180,E1 23123.923,E2 23123.923} C_VEL
LIN {X 0,Y 472.548,Z 550.612,A -85,B 0,C 180,E1 23121.604,E2 23121.604} C_VEL
LIN {X 0,Y 472.99,Z 544.039,A -85,B 0,C 180,E1 23119.402,E2 23119.402} C_VEL
LIN {X 0,Y 473.681,Z 535.655,A -85,B 0,C 180,E1 23117.215,E2 23117.215} C_VEL
LIN {X 0,Y 474.56,Z 526.207,A -85,B 0,C 180,E1 23115.229,E2 23115.229} C_VEL
LIN {X 0,Y 475.704,Z 514.773,A -85,B 0,C 180,E1 23113.264,E2 23113.264} C_VEL
LIN {X 0,Y 476.966,Z 502.696,A -85,B 0,C 180,E1 23111.546,E2 23111.546} C_VEL
LIN {X 0,Y 478.345,Z 489.238,A -85,B 0,C 180,E1 23109.952,E2 23109.952} C_VEL
LIN {X 0,Y 479.813,Z 474.219,A -85,B 0,C 180,E1 23108.484,E2 23108.484} C_VEL
LIN {X 0,Y 481.165,Z 459.02,A -85,B 0,C 180,E1 23107.262,E2 23107.262} C_VEL
LIN {X 0,Y 482.48,Z 442.061,A -85,B 0,C 180,E1 23106.164,E2 23106.164} C_VEL
LIN {X 0,Y 483.582,Z 424.563,A -85,B 0,C 180,E1 23105.28,E2 23105.28} C_VEL
LIN {X 0,Y 484.425,Z 406.193,A -85,B 0,C 180,E1 23104.592,E2 23104.592} C_VEL
LIN {X 0,Y 484.979,Z 387.307,A -85,B 0,C 180,E1 23104.117,E2 23104.117} C_VEL
LIN {X 0,Y 486.78,Z 195.159,A -85,B 0,C 180,E1 23101.284,E2 23101.284} C_VEL
LIN {X 0,Y 482.864,Z 173.768,A -85,B 0,C 180,E1 23100.64,E2 23100.64} C_VEL
LIN {X 0,Y 484.768,Z 143.484,A -85,B 0,C 180,E1 23097.811,E2 23097.811} C_VEL
LIN {X 0,Y 478.18,Z 124.773,A -85,B 0,C 180,E1 23095.337,E2 23095.337} C_VEL
LIN {X 0,Y 472.951,Z 110.583,A -85,B 0,C 180,E1 23093.328,E2 23093.328} C_VEL
LIN {X 0,Y 472.949,Z 110.553,A -85,B 0,C 180,E1 23089.69,E2 23089.69} C_VEL
LIN {X 0,Y 472.94,Z 110.569,A -85,B 0,C 180,E1 23086.097,E2 23086.097} C_VEL
LIN {X 0,Y 472.939,Z 110.57,A -85,B 0,C 180,E1 23082.409,E2 23082.409} C_VEL
LIN {X 0,Y 472.944,Z 110.572,A -85,B 0,C 180,E1 23078.729,E2 23078.729} C_VEL
LIN {X 0,Y 472.951,Z 110.575,A -85,B 0,C 180,E1 23075.005,E2 23075.005} C_VEL
LIN {X 0,Y 481.845,Z 136.67,A -85,B 0,C 180,E1 23072.088,E2 23072.088} C_VEL
LIN {X 0,Y 482.7,Z 139.959,A -85,B 0,C 180,E1 23071.745,E2 23071.745} C_VEL
LIN {X 0,Y 481.464,Z 178.211,A -85,B 0,C 180,E1 23068.532,E2 23068.532} C_VEL
LIN {X 0,Y 481.487,Z 181.412,A -85,B 0,C 180,E1 23068.299,E2 23068.299} C_VEL
LIN {X 0,Y 483.597,Z 195.792,A -85,B 0,C 180,E1 23067.905,E2 23067.905} C_VEL
LIN {X 0,Y 480.257,Z 391.264,A -85,B 0,C 180,E1 23064.57,E2 23064.57} C_VEL
LIN {X 0,Y 479.756,Z 410.679,A -85,B 0,C 180,E1 23064.012,E2 23064.012} C_VEL
LIN {X 0,Y 479.05,Z 429.499,A -85,B 0,C 180,E1 23063.234,E2 23063.234} C_VEL
LIN {X 0,Y 478.222,Z 447.075,A -85,B 0,C 180,E1 23062.278,E2 23062.278} C_VEL
LIN {X 0,Y 477.306,Z 463.994,A -85,B 0,C 180,E1 23061.119,E2 23061.119} C_VEL
LIN {X 0,Y 476.339,Z 480.192,A -85,B 0,C 180,E1 23059.752,E2 23059.752} C_VEL
LIN {X 0,Y 475.383,Z 495.292,A -85,B 0,C 180,E1 23058.2,E2 23058.2} C_VEL
LIN {X 0,Y 474.521,Z 508.842,A -85,B 0,C 180,E1 23056.517,E2 23056.517} C_VEL
LIN {X 0,Y 473.803,Z 520.374,A -85,B 0,C 180,E1 23054.794,E2 23054.794} C_VEL
LIN {X 0,Y 473.21,Z 530.675,A -85,B 0,C 180,E1 23052.943,E2 23052.943} C_VEL
LIN {X 0,Y 472.755,Z 539.647,A -85,B 0,C 180,E1 23050.973,E2 23050.973} C_VEL
LIN {X 0,Y 472.436,Z 547.227,A -85,B 0,C 180,E1 23048.888,E2 23048.888} C_VEL
LIN {X 0,Y 472.241,Z 553.333,A -85,B 0,C 180,E1 23046.687,E2 23046.687} C_VEL
LIN {X 0,Y 472.129,Z 557.639,A -85,B 0,C 180,E1 23044.494,E2 23044.494} C_VEL
LIN {X 0,Y 472.094,Z 560.375,A -85,B 0,C 180,E1 23042.185,E2 23042.185} C_VEL
LIN {X 0,Y 472.091,Z 561.296,A -85,B 0,C 180,E1 23039.879,E2 23039.879} C_VEL
LIN {X 0,Y 472.107,Z 560.435,A -85,B 0,C 180,E1 23037.573,E2 23037.573} C_VEL
LIN {X 0,Y 472.166,Z 557.974,A -85,B 0,C 180,E1 23035.385,E2 23035.385} C_VEL
LIN {X 0,Y 472.295,Z 553.755,A -85,B 0,C 180,E1 23033.164,E2 23033.164} C_VEL
LIN {X 0,Y 472.515,Z 547.842,A -85,B 0,C 180,E1 23030.991,E2 23030.991} C_VEL
LIN {X 0,Y 472.866,Z 540.106,A -85,B 0,C 180,E1 23028.849,E2 23028.849} C_VEL
LIN {X 0,Y 473.371,Z 530.801,A -85,B 0,C 180,E1 23026.814,E2 23026.814} C_VEL
LIN {X 0,Y 473.988,Z 520.357,A -85,B 0,C 180,E1 23024.962,E2 23024.962} C_VEL
LIN {X 0,Y 474.719,Z 508.486,A -85,B 0,C 180,E1 23023.229,E2 23023.229} C_VEL
LIN {X 0,Y 475.572,Z 494.599,A -85,B 0,C 180,E1 23021.554,E2 23021.554} C_VEL
LIN {X 0,Y 476.449,Z 479.773,A -85,B 0,C 180,E1 23020.079,E2 23020.079} C_VEL
LIN {X 0,Y 477.305,Z 463.763,A -85,B 0,C 180,E1 23018.779,E2 23018.779} C_VEL
LIN {X 0,Y 478.077,Z 447.122,A -85,B 0,C 180,E1 23017.692,E2 23017.692} C_VEL
LIN {X 0,Y 478.774,Z 428.876,A -85,B 0,C 180,E1 23016.753,E2 23016.753} C_VEL
LIN {X 0,Y 479.301,Z 409.96,A -85,B 0,C 180,E1 23016.027,E2 23016.027} C_VEL
LIN {X 0,Y 479.653,Z 390.474,A -85,B 0,C 180,E1 23015.516,E2 23015.516} C_VEL
LIN {X 0,Y 481.664,Z 281.453,A -85,B 0,C 180,E1 23013.568,E2 23013.568} C_VEL
LIN {X 0,Y 484.093,Z 193.69,A -85,B 0,C 180,E1 23011.831,E2 23011.831} C_VEL
LIN {X 0,Y 483.269,Z 188.148,A -85,B 0,C 180,E1 23011.619,E2 23011.619} C_VEL
LIN {X 0,Y 483.971,Z 149.474,A -85,B 0,C 180,E1 23008.566,E2 23008.566} C_VEL
LIN {X 0,Y 483.912,Z 138.421,A -85,B 0,C 180,E1 23007.681,E2 23007.681} C_VEL
LIN {X 0,Y 479.445,Z 125.286,A -85,B 0,C 180,E1 23006.208,E2 23006.208} C_VEL
LIN {X 0,Y 474.644,Z 114.631,A -85,B 0,C 180,E1 23004.82,E2 23004.82} C_VEL
LIN {X 0,Y 473.064,Z 111.434,A -85,B 0,C 180,E1 23004.377,E2 23004.377} C_VEL
LIN {X 0,Y 472.912,Z 110.579,A -85,B 0,C 180,E1 23004.28,E2 23004.28} C_VEL
LIN {X 0,Y 472.901,Z 110.58,A -85,B 0,C 180,E1 23000.633,E2 23000.633} C_VEL
LIN {X 0,Y 472.906,Z 110.58,A -85,B 0,C 180,E1 22997.094,E2 22997.094} C_VEL
LIN {X 0,Y 472.927,Z 110.577,A -85,B 0,C 180,E1 22993.517,E2 22993.517} C_VEL
LIN {X 0,Y 472.896,Z 110.689,A -85,B 0,C 180,E1 22990.572,E2 22990.572} C_VEL
LIN {X 0,Y 473.991,Z 113.722,A -85,B 0,C 180,E1 22990.203,E2 22990.203} C_VEL
LIN {X 0,Y 481.741,Z 132.238,A -85,B 0,C 180,E1 22987.937,E2 22987.937} C_VEL
LIN {X 0,Y 487.376,Z 147.069,A -85,B 0,C 180,E1 22986.27,E2 22986.27} C_VEL
LIN {X 0,Y 486.396,Z 164.483,A -85,B 0,C 180,E1 22984.984,E2 22984.984} C_VEL
LIN {X 0,Y 489.166,Z 185.258,A -85,B 0,C 180,E1 22984.412,E2 22984.412} C_VEL
LIN {X 0,Y 484.995,Z 423.554,A -85,B 0,C 180,E1 22980.49,E2 22980.49} C_VEL
LIN {X 0,Y 484.144,Z 445.151,A -85,B 0,C 180,E1 22979.918,E2 22979.918} C_VEL
LIN {X 0,Y 483.036,Z 466.649,A -85,B 0,C 180,E1 22979.107,E2 22979.107} C_VEL
LIN {X 0,Y 481.779,Z 486.875,A -85,B 0,C 180,E1 22978.107,E2 22978.107} C_VEL
LIN {X 0,Y 480.454,Z 505.937,A -85,B 0,C 180,E1 22976.93,E2 22976.93} C_VEL
LIN {X 0,Y 479.126,Z 523.825,A -85,B 0,C 180,E1 22975.594,E2 22975.594} C_VEL
LIN {X 0,Y 477.686,Z 542.1,A -85,B 0,C 180,E1 22973.959,E2 22973.959} C_VEL
LIN {X 0,Y 476.426,Z 558.061,A -85,B 0,C 180,E1 22972.255,E2 22972.255} C_VEL
LIN {X 0,Y 475.288,Z 572.528,A -85,B 0,C 180,E1 22970.44,E2 22970.44} C_VEL
LIN {X 0,Y 474.281,Z 586.057,A -85,B 0,C 180,E1 22968.435,E2 22968.435} C_VEL
LIN {X 0,Y 473.454,Z 598.097,A -85,B 0,C 180,E1 22966.313,E2 22966.313} C_VEL
LIN {X 0,Y 472.85,Z 608.168,A -85,B 0,C 180,E1 22964.199,E2 22964.199} C_VEL
LIN {X 0,Y 472.399,Z 617.404,A -85,B 0,C 180,E1 22961.848,E2 22961.848} C_VEL
LIN {X 0,Y 472.142,Z 624.366,A -85,B 0,C 180,E1 22959.632,E2 22959.632} C_VEL
LIN {X 0,Y 471.99,Z 630.003,A -85,B 0,C 180,E1 22957.181,E2 22957.181} C_VEL
LIN {X 0,Y 471.922,Z 633.925,A -85,B 0,C 180,E1 22954.74,E2 22954.74} C_VEL
LIN {X 0,Y 471.906,Z 636.302,A -85,B 0,C 180,E1 22952.186,E2 22952.186} C_VEL
LIN {X 0,Y 471.905,Z 636.961,A -85,B 0,C 180,E1 22949.758,E2 22949.758} C_VEL
LIN {X 0,Y 471.908,Z 636.03,A -85,B 0,C 180,E1 22947.329,E2 22947.329} C_VEL
LIN {X 0,Y 471.929,Z 633.446,A -85,B 0,C 180,E1 22944.896,E2 22944.896} C_VEL
LIN {X 0,Y 471.999,Z 629.245,A -85,B 0,C 180,E1 22942.454,E2 22942.454} C_VEL
LIN {X 0,Y 472.161,Z 623.666,A -85,B 0,C 180,E1 22940.124,E2 22940.124} C_VEL
LIN {X 0,Y 472.434,Z 616.536,A -85,B 0,C 180,E1 22937.897,E2 22937.897} C_VEL
LIN {X 0,Y 472.911,Z 607.108,A -85,B 0,C 180,E1 22935.554,E2 22935.554} C_VEL
LIN {X 0,Y 473.577,Z 596.124,A -85,B 0,C 180,E1 22933.314,E2 22933.314} C_VEL
LIN {X 0,Y 474.486,Z 583.147,A -85,B 0,C 180,E1 22931.112,E2 22931.112} C_VEL
LIN {X 0,Y 475.572,Z 568.731,A -85,B 0,C 180,E1 22929.06,E2 22929.06} C_VEL
LIN {X 0,Y 476.778,Z 553.615,A -85,B 0,C 180,E1 22927.238,E2 22927.238} C_VEL
LIN {X 0,Y 478.091,Z 537.315,A -85,B 0,C 180,E1 22925.576,E2 22925.576} C_VEL
LIN {X 0,Y 479.491,Z 519.213,A -85,B 0,C 180,E1 22924.031,E2 22924.031} C_VEL
LIN {X 0,Y 480.827,Z 500.736,A -85,B 0,C 180,E1 22922.724,E2 22922.724} C_VEL
LIN {X 0,Y 482.08,Z 482.185,A -85,B 0,C 180,E1 22921.644,E2 22921.644} C_VEL
LIN {X 0,Y 483.274,Z 461.756,A -85,B 0,C 180,E1 22920.692,E2 22920.692} C_VEL
LIN {X 0,Y 484.345,Z 440.435,A -85,B 0,C 180,E1 22919.944,E2 22919.944} C_VEL
LIN {X 0,Y 485.092,Z 419.758,A -85,B 0,C 180,E1 22919.437,E2 22919.437} C_VEL
LIN {X 0,Y 489.187,Z 183.891,A -85,B 0,C 180,E1 22915.564,E2 22915.564} C_VEL
LIN {X 0,Y 486.339,Z 163.383,A -85,B 0,C 180,E1 22914.964,E2 22914.964} C_VEL
LIN {X 0,Y 487.297,Z 146.646,A -85,B 0,C 180,E1 22913.693,E2 22913.693} C_VEL
LIN {X 0,Y 478.735,Z 124.636,A -85,B 0,C 180,E1 22911.171,E2 22911.171} C_VEL
LIN {X 0,Y 473.721,Z 113.185,A -85,B 0,C 180,E1 22909.729,E2 22909.729} C_VEL
LIN {X 0,Y 472.906,Z 110.576,A -85,B 0,C 180,E1 22909.412,E2 22909.412} C_VEL
LIN {X 0,Y 472.941,Z 110.568,A -85,B 0,C 180,E1 22905.93,E2 22905.93} C_VEL
LIN {X 0,Y 472.946,Z 110.57,A -85,B 0,C 180,E1 22902.243,E2 22902.243} C_VEL
LIN {X 0,Y 472.905,Z 110.536,A -85,B 0,C 180,E1 22898.725,E2 22898.725} C_VEL
LIN {X 0,Y 472.895,Z 110.577,A -85,B 0,C 180,E1 22895.255,E2 22895.255} C_VEL
LIN {X 0,Y 472.917,Z 110.575,A -85,B 0,C 180,E1 22891.765,E2 22891.765} C_VEL
LIN {X 0,Y 472.951,Z 110.562,A -85,B 0,C 180,E1 22888.265,E2 22888.265} C_VEL
LIN {X 0,Y 472.921,Z 110.568,A -85,B 0,C 180,E1 22884.614,E2 22884.614} C_VEL
LIN {X 0,Y 472.893,Z 110.576,A -85,B 0,C 180,E1 22881.187,E2 22881.187} C_VEL
LIN {X 0,Y 472.894,Z 110.574,A -85,B 0,C 180,E1 22877.532,E2 22877.532} C_VEL
LIN {X 0,Y 472.927,Z 110.562,A -85,B 0,C 180,E1 22874.071,E2 22874.071} C_VEL
LIN {X 0,Y 472.937,Z 110.574,A -85,B 0,C 180,E1 22870.475,E2 22870.475} C_VEL
LIN {X 0,Y 472.901,Z 110.559,A -85,B 0,C 180,E1 22866.922,E2 22866.922} C_VEL
LIN {X 0,Y 472.887,Z 110.576,A -85,B 0,C 180,E1 22863.394,E2 22863.394} C_VEL
LIN {X 0,Y 472.892,Z 110.573,A -85,B 0,C 180,E1 22859.757,E2 22859.757} C_VEL
LIN {X 0,Y 472.924,Z 110.568,A -85,B 0,C 180,E1 22856.242,E2 22856.242} C_VEL
LIN {X 0,Y 472.938,Z 110.569,A -85,B 0,C 180,E1 22852.59,E2 22852.59} C_VEL
LIN {X 0,Y 472.899,Z 110.567,A -85,B 0,C 180,E1 22849.03,E2 22849.03} C_VEL
